# B&R Automation Studio project FlyingSaw2023
Automation Studio 4.12.2.93; technology packages: mapp 5.22.1, mappCockpit 5.22.0, mappMotion 5.22.2, mappView 5.22.1

## Configuration Config1

CPU X20CP3586, AutomationRuntime F4.93, Build 4.1.2, Safety 0.0, Vc V4.72.0

### Task classes (Cpu.sw)
```
Cyclic#1 (cycle 2000 us, tolerance 0 us):
  Saw_P <- Libraries.Saw.Saw_P.prg
  Main <- Main.prg
  ConveyorAx <- ConveyorAxis.prg
  ParallelAx <- ParallelAxis.prg
  Perpendicu <- PerpendicularAxis.prg
  Alarm <- Alarm.prg
  Recipe <- Recipe.prg
  Program <- (binary)
DataObjects: McAcpSys
NcDataObjects: McDriveLog
Binaries: udbdef, FWRules, TCData, arsvcreg, McAcpDrv, arflatprv, arcoal, McAcpSim, mvLoader, mCoWebSc, sysconf, Role, User, iomap, ashwd, asfw, arconfig, ashwac, Config_1, Config_2, Settings, Config, Config_3, McProfGen
Libraries: AsBrStr, AsTCP, standard, runtime, Saw_L, operator, McBase, CoTrace, AsZip, FileIO, MpAxis, McAxis, MpBase, McAcpAx, MpAlarmX, astime, MpServer, MpRecipe, sys_lib, asieccon, powerlnk, asepl, arssl, dataobj, aruser
```

### Hardware
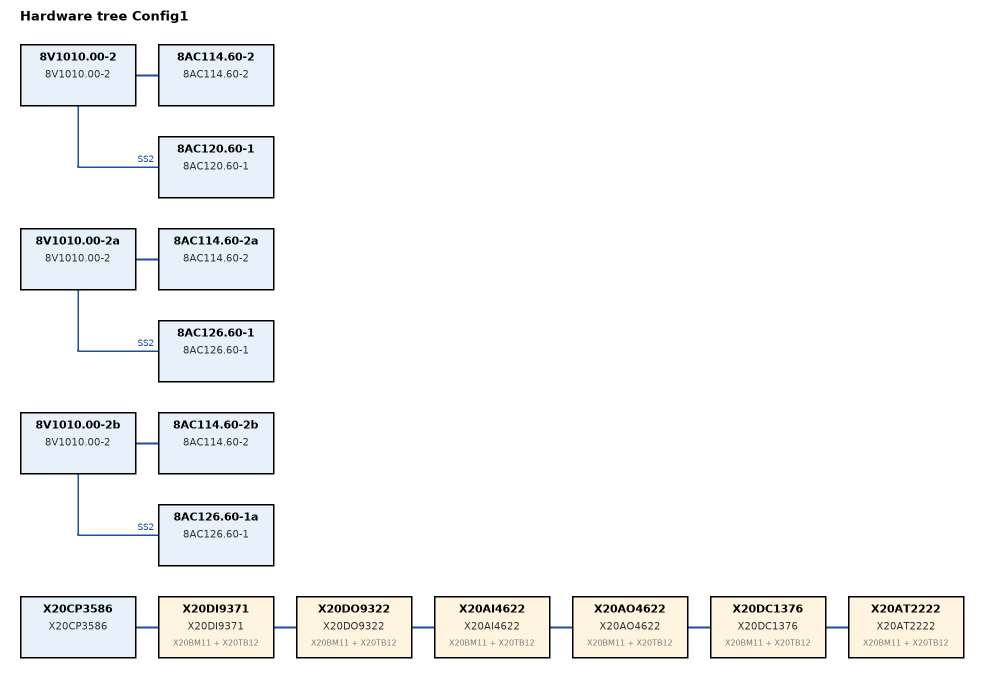
```
8AC114.60-2 : 8AC114.60-2 v1.0.0.8  [SS -> 8V1010.00-2.SS1; PLK1 -> X20CP3586.IF3 (NodeNumber=1) [Cable Type=PowerlinkCable, Length=10, Version=1.0.0.3]; PLK2 -> 8AC114.60-2a.PLK1 (NodeNumber=1) [Cable Type=PowerlinkCable, Length=10, Version=1.0.0.3]]
8AC114.60-2a : 8AC114.60-2 v1.0.0.8  [SS -> 8V1010.00-2a.SS1; PLK1 -> 8AC114.60-2.PLK2 (NodeNumber=2) [Cable Type=PowerlinkCable, Length=10, Version=1.0.0.3]; PLK2 -> 8AC114.60-2b.PLK1 (NodeNumber=2) [Cable Type=PowerlinkCable, Length=10, Version=1.0.0.3]]
8AC114.60-2b : 8AC114.60-2 v1.0.0.8  [SS -> 8V1010.00-2b.SS1; PLK1 -> 8AC114.60-2a.PLK2 (NodeNumber=3) [Cable Type=PowerlinkCable, Length=10, Version=1.0.0.3]]
8AC120.60-1 : 8AC120.60-1 v2.2.0.0  [SS -> 8V1010.00-2.SS2]
  PlugInType = Encoder
  McAcoposTypeID = AcoposPlugInConfig
8AC126.60-1 : 8AC126.60-1 v2.2.0.0  [SS -> 8V1010.00-2a.SS2]
  PlugInType = Encoder
  McAcoposTypeID = AcoposPlugInConfig
8AC126.60-1a : 8AC126.60-1 v2.2.0.0  [SS -> 8V1010.00-2b.SS2]
  PlugInType = Encoder
  McAcoposTypeID = AcoposPlugInConfig
8V1010.00-2 : 8V1010.00-2 v2.2.0.0
  DriveConfiguration/Module:
    McAcoposTypeID = AcoposConfig
    ActivateACOPOSSimulationOnPLC = 0
    PowerSupply = ETA
  DriveConfiguration/Channel[1]/RealAxis:
    AxisReference = gParallelAxis
    MechanicalElementsIsInvisible = 0
  DriveConfiguration/Channel[1]/RealAxis/MechanicalElements/Gearbox:
    InputIsReadOnly = 0
    Input = 1
    OutputIsReadOnly = 0
    Output = 1
  DriveConfiguration/Channel[1]/RealAxis/MechanicalElements/RotaryToLinearTransformation:
    ReferenceDistanceIsReadOnly = 0
    ReferenceDistance = 1.6
  DriveConfiguration/Channel[1]/RealAxis/Controller:
    ModeIsReadOnly = 0
    Mode = PositionController
  DriveConfiguration/Channel[1]/RealAxis/Controller/Mode/Position:
    ProportionalGain = 907
    IntegrationTime = 0.0
    PredictionTime = 0.0004
    TotalDelayTime = 0.0004
  DriveConfiguration/Channel[1]/RealAxis/Controller/Mode/Speed:
    ProportionalGainIsReadOnly = 0
    ProportionalGain = 0.05
    IntegrationTimeIsReadOnly = 0
    IntegrationTime = 0.0
    FilterTimeIsReadOnly = 0
    FilterTime = 0.0
  DriveConfiguration/Channel[1]/RealAxis/Controller/Mode/LoopFilters:
    LoopFilterXIsReadOnly = 0
    LoopFilter1 = NotUsed
    LoopFilter2 = NotUsed
    LoopFilter3 = NotUsed
  DriveConfiguration/Channel[1]/RealAxis/Homing:
    ModeIsReadOnly = 0
    Mode = LimitSwitch
  DriveConfiguration/Channel[1]/RealAxis/Homing/Mode:
    Position = -0.8
    StartVelocity = 0.5
    HomingVelocity = 0.05
    Acceleration = 50.0
    SwitchEdge = Negative
    HomingDirection = Positive
    KeepDirection = No
    ReferencePulse = NotUsed
  DriveConfiguration/Channel[1]/RealAxis/Homing:
    RestorePositionVariable = 
  DriveConfiguration/Channel[1]/RealAxis/StopReaction:
    QuickstopIsReadOnly = 0
    Quickstop = DecelerationLimit
    DriveErrorIsReadOnly = 0
    DriveError = DecelerationLimit
  DriveConfiguration/Channel[1]/RealAxis/MovementErrorLimits:
    PositionError = 10
    VelocityErrorMonitoring = NotUsed
  DriveConfiguration/Channel[1]/RealAxis:
    JerkFilterIsReadOnly = 0
    JerkFilter = NotUsed
    ZeroVibrationFilter = NotUsed
  DriveConfiguration/Channel[1]/RealAxis/DigitalInputs/HomingSwitch:
    SourceIsReadOnly = 0
    Source = X1Ref
    Level = High
  DriveConfiguration/Channel[1]/RealAxis/DigitalInputs/PositiveLimitSwitch:
    Source = Variable
  DriveConfiguration/Channel[1]/RealAxis/DigitalInputs/PositiveLimitSwitch/Source:
    PVmapping = ::Saw_SimInputs.diDriveParallelAtFront
  DriveConfiguration/Channel[1]/RealAxis/DigitalInputs/PositiveLimitSwitch:
    Level = High
  DriveConfiguration/Channel[1]/RealAxis/DigitalInputs/NegativeLimitSwitch:
    Source = Variable
  DriveConfiguration/Channel[1]/RealAxis/DigitalInputs/NegativeLimitSwitch/Source:
    PVmapping = ::Saw_SimInputs.diDriveParallelAtBack
  DriveConfiguration/Channel[1]/RealAxis/DigitalInputs/NegativeLimitSwitch:
    Level = High
  DriveConfiguration/Channel[1]/RealAxis/DigitalInputs/Trigger1:
    Source = X1Trigger1
    Level = High
  DriveConfiguration/Channel[1]/RealAxis/DigitalInputs/Trigger2:
    Source = X1Trigger2
    Level = High
  DriveConfiguration/Channel[1]/RealAxis/DigitalInputs/Quickstop:
    Input = Trigger2
  DriveConfiguration/Channel[1]/RealAxis/Simulation:
    SimulationModeOnPLC = SetValueGeneration
    SimulationModeOnACOPOS = NotUsed
  DriveConfiguration/Channel[1]/RealAxis/AxisFeatures:
    FeatureRef[1] = CamAutomatParallel
  DriveConfiguration/Channel[1]:
    ExternalEncoderAxis = NotUsed
8V1010.00-2a : 8V1010.00-2 v2.2.0.0
  DriveConfiguration/Module:
    McAcoposTypeID = AcoposConfig
    ActivateACOPOSSimulationOnPLC = 0
    PowerSupply = ETA
  DriveConfiguration/Channel[1]/RealAxis:
    AxisReference = gPerpendicularAxis
    MechanicalElementsIsInvisible = 0
  DriveConfiguration/Channel[1]/RealAxis/MechanicalElements/Gearbox:
    InputIsReadOnly = 0
    Input = 1
    OutputIsReadOnly = 0
    Output = 1
  DriveConfiguration/Channel[1]/RealAxis/MechanicalElements/RotaryToLinearTransformation:
    ReferenceDistanceIsReadOnly = 0
    ReferenceDistance = 1.6
  DriveConfiguration/Channel[1]/RealAxis/Controller:
    ModeIsReadOnly = 0
    Mode = PositionController
  DriveConfiguration/Channel[1]/RealAxis/Controller/Mode/Position:
    ProportionalGain = 215
    IntegrationTime = 0.0
    PredictionTime = 0.0004
    TotalDelayTime = 0.0004
  DriveConfiguration/Channel[1]/RealAxis/Controller/Mode/Speed:
    ProportionalGainIsReadOnly = 0
    ProportionalGain = 0.041
    IntegrationTimeIsReadOnly = 0
    IntegrationTime = 0.0
    FilterTimeIsReadOnly = 0
    FilterTime = 0.0
  DriveConfiguration/Channel[1]/RealAxis/Controller/Mode/LoopFilters:
    LoopFilterXIsReadOnly = 0
    LoopFilter1 = NotUsed
    LoopFilter2 = NotUsed
    LoopFilter3 = NotUsed
  DriveConfiguration/Channel[1]/RealAxis/Homing:
    ModeIsReadOnly = 0
    Mode = LimitSwitch
  DriveConfiguration/Channel[1]/RealAxis/Homing/Mode:
    Position = -0.6
    StartVelocity = 0.5
    HomingVelocity = 0.05
    Acceleration = 50.0
    SwitchEdge = Negative
    HomingDirection = Positive
    KeepDirection = No
    ReferencePulse = NotUsed
  DriveConfiguration/Channel[1]/RealAxis/Homing:
    RestorePositionVariable = 
  DriveConfiguration/Channel[1]/RealAxis/StopReaction:
    QuickstopIsReadOnly = 0
    Quickstop = DecelerationLimit
    DriveErrorIsReadOnly = 0
    DriveError = DecelerationLimit
  DriveConfiguration/Channel[1]/RealAxis/MovementErrorLimits:
    PositionError = 10
    VelocityErrorMonitoring = NotUsed
  DriveConfiguration/Channel[1]/RealAxis:
    JerkFilterIsReadOnly = 0
    JerkFilter = NotUsed
    ZeroVibrationFilter = NotUsed
  DriveConfiguration/Channel[1]/RealAxis/DigitalInputs/HomingSwitch:
    SourceIsReadOnly = 0
    Source = X1Ref
    Level = High
  DriveConfiguration/Channel[1]/RealAxis/DigitalInputs/PositiveLimitSwitch:
    Source = Variable
  DriveConfiguration/Channel[1]/RealAxis/DigitalInputs/PositiveLimitSwitch/Source:
    PVmapping = ::Saw_SimInputs.diDriveCutAtFront
  DriveConfiguration/Channel[1]/RealAxis/DigitalInputs/PositiveLimitSwitch:
    Level = High
  DriveConfiguration/Channel[1]/RealAxis/DigitalInputs/NegativeLimitSwitch:
    Source = Variable
  DriveConfiguration/Channel[1]/RealAxis/DigitalInputs/NegativeLimitSwitch/Source:
    PVmapping = ::Saw_SimInputs.diDriveCutAtBack
  DriveConfiguration/Channel[1]/RealAxis/DigitalInputs/NegativeLimitSwitch:
    Level = High
  DriveConfiguration/Channel[1]/RealAxis/DigitalInputs/Trigger1:
    Source = X1Trigger1
    Level = High
  DriveConfiguration/Channel[1]/RealAxis/DigitalInputs/Trigger2:
    Source = X1Trigger2
    Level = High
  DriveConfiguration/Channel[1]/RealAxis/DigitalInputs/Quickstop:
    Input = Trigger2
  DriveConfiguration/Channel[1]/RealAxis/Simulation:
    SimulationModeOnPLC = SetValueGeneration
    SimulationModeOnACOPOS = NotUsed
  DriveConfiguration/Channel[1]/RealAxis/AxisFeatures:
    FeatureRef[1] = CamAutomatPerpendicular
  DriveConfiguration/Channel[1]:
    ExternalEncoderAxis = NotUsed
8V1010.00-2b : 8V1010.00-2 v2.2.0.0
  DriveConfiguration/Module:
    McAcoposTypeID = AcoposConfig
    ActivateACOPOSSimulationOnPLC = 1
    PowerSupply = ETA
  DriveConfiguration/Channel[1]/RealAxis:
    AxisReference = gConveyorAxis
    MechanicalElementsIsInvisible = 0
  DriveConfiguration/Channel[1]/RealAxis/MechanicalElements/Gearbox:
    InputIsReadOnly = 0
    Input = 1
    OutputIsReadOnly = 0
    Output = 1
  DriveConfiguration/Channel[1]/RealAxis/MechanicalElements/RotaryToLinearTransformation:
    ReferenceDistanceIsReadOnly = 0
    ReferenceDistance = 1
  DriveConfiguration/Channel[1]/RealAxis/Controller:
    ModeIsReadOnly = 0
    Mode = PositionController
  DriveConfiguration/Channel[1]/RealAxis/Controller/Mode/Position:
    ProportionalGain = 50.0
    IntegrationTime = 0.0
    PredictionTime = 0.0004
    TotalDelayTime = 0.0004
  DriveConfiguration/Channel[1]/RealAxis/Controller/Mode/Speed:
    ProportionalGainIsReadOnly = 0
    ProportionalGain = 2.0
    IntegrationTimeIsReadOnly = 0
    IntegrationTime = 0.0
    FilterTimeIsReadOnly = 0
    FilterTime = 0.0
  DriveConfiguration/Channel[1]/RealAxis/Controller/Mode/LoopFilters:
    LoopFilterXIsReadOnly = 0
    LoopFilter1 = NotUsed
    LoopFilter2 = NotUsed
    LoopFilter3 = NotUsed
  DriveConfiguration/Channel[1]/RealAxis/Homing:
    ModeIsReadOnly = 0
    Mode = Direct
  DriveConfiguration/Channel[1]/RealAxis/Homing/Mode:
    Position = 0.0
    ReferencePulse = NotUsed
  DriveConfiguration/Channel[1]/RealAxis/Homing:
    RestorePositionVariable = 
  DriveConfiguration/Channel[1]/RealAxis/StopReaction:
    QuickstopIsReadOnly = 0
    Quickstop = DecelerationLimit
    DriveErrorIsReadOnly = 0
    DriveError = DecelerationLimit
  DriveConfiguration/Channel[1]/RealAxis/MovementErrorLimits:
    PositionError = 1.0
    VelocityErrorMonitoring = Automatic1
  DriveConfiguration/Channel[1]/RealAxis:
    JerkFilterIsReadOnly = 0
    JerkFilter = NotUsed
    ZeroVibrationFilter = NotUsed
  DriveConfiguration/Channel[1]/RealAxis/DigitalInputs/HomingSwitch:
    SourceIsReadOnly = 0
    Source = X1Ref
    Level = High
  DriveConfiguration/Channel[1]/RealAxis/DigitalInputs/PositiveLimitSwitch:
    Source = X1PosLim
    Level = High
  DriveConfiguration/Channel[1]/RealAxis/DigitalInputs/NegativeLimitSwitch:
    Source = X1NegLim
    Level = High
  DriveConfiguration/Channel[1]/RealAxis/DigitalInputs/Trigger1:
    Source = X1Trigger1
    Level = High
  DriveConfiguration/Channel[1]/RealAxis/DigitalInputs/Trigger2:
    Source = X1Trigger2
    Level = High
  DriveConfiguration/Channel[1]/RealAxis/DigitalInputs/Quickstop:
    Input = Trigger2
  DriveConfiguration/Channel[1]/RealAxis/Simulation:
    SimulationModeOnPLC = SetValueGeneration
    SimulationModeOnACOPOS = NotUsed
  DriveConfiguration/Channel[1]/RealAxis/AxisFeatures:
    FeatureRef[1] = Feature_CamAutomat
  DriveConfiguration/Channel[1]:
    ExternalEncoderAxis = NotUsed
X20AI4622 : X20AI4622 v1.2.0.0  [SS1 -> X20TB12b.SS; SL -> X20BM11b.SL1]
X20AO4622 : X20AO4622 v1.3.0.0  [SS1 -> X20TB12c.SS; SL -> X20BM11c.SL1]
X20AT2222 : X20AT2222 v1.4.0.0  [SS1 -> X20TB12e.SS; SL -> X20BM11e.SL1]
X20BM11 : X20BM11 v1.1.0.0  [X2X1 -> X20CP3586.IF6]
X20BM11a : X20BM11 v1.1.0.0  [X2X1 -> X20BM11.X2X2]
X20BM11b : X20BM11 v1.1.0.0  [X2X1 -> X20BM11a.X2X2]
X20BM11c : X20BM11 v1.1.0.0  [X2X1 -> X20BM11b.X2X2]
X20BM11d : X20BM11 v1.1.0.0  [X2X1 -> X20BM11c.X2X2]
X20BM11e : X20BM11 v1.1.0.0  [X2X1 -> X20BM11d.X2X2]
X20CP3586 : X20CP3586 v1.10.0.0
  Connector IF2:
    ActivateDevice = 1
    Mode = Manual
    InternetAddress = 10.0.0.2
    SubnetMask = 255.255.255.0
    ActivateSnmp = 2
  Connector IF3:
    DNAConfiguration = manual
    Channel1
    ChannelID1 = McAcpBroadcast
    ChannelType1 = OCTET[96]
  ConfigurationID = FlyingSaw2023_Config1
  UserPartitionSize = 0
  Simulation = 1
  TimerDeviceType = EPLX2X
  TimerDevice = X20CP3586.IF3
  TaskClassIdleTime = 2000
  Cyclic1Duration = 2000
  Cyclic1Tolerance = 0
  FileDevice1
  FileDeviceName1 = USER
  FileDevicePath1 = C:\temp
  ActivateOpcUa = 1
  OpcUaInformationModels_PV_Version = 1
X20DC1376 : X20DC1376 v1.3.0.0  [SS1 -> X20TB12d.SS; SL -> X20BM11d.SL1]
X20DI9371 : X20DI9371 v1.4.0.0  [SS1 -> X20TB12.SS; SL -> X20BM11.SL1]
X20DO9322 : X20DO9322 v1.5.0.0  [SS1 -> X20TB12a.SS; SL -> X20BM11a.SL1]
X20TB12 : X20TB12 v1.0.0.0
X20TB12a : X20TB12 v1.0.0.0
X20TB12b : X20TB12 v1.0.0.0
X20TB12c : X20TB12 v1.0.0.0
X20TB12d : X20TB12 v1.0.0.0
X20TB12e : X20TB12 v1.0.0.0
```

### IoMap.iom - X20CP3586/IoMap.iom
```iecst
VAR_CONFIG
	::Main:SawLeft AT %IX."X20DI9371".DigitalInput01;
	::Main:SawRight AT %IX."X20DI9371".DigitalInput02;
	::Main:SawRunAxis AT %IX."X20DI9371".DigitalInput06;
	::Tasmociag:MpAxisConveyor.MoveVelocity AT %QX."X20DO9322".DigitalOutput01;
	::Main:RunConveyor AT %IX."X20DI9371".DigitalInput05;
	::Main:SawForward AT %IX."X20DI9371".DigitalInput03;
	::Main:SawBackward AT %IX."X20DI9371".DigitalInput04;
	::OsRownoleg:MpAxisParallel.Power AT %QX."X20DO9322".DigitalOutput02;
	::OsRownoleg:MpAxisParallel.Power AT %QX."X20DO9322".DigitalOutput03;
END_VAR
```

### Config_1.axis - X20CP3586/mappMotion/Config_1.axis
```
Element gPerpendicularAxis (Type=axis)
  BaseTypeIsReadOnly = 0
  BaseType = LinearBounded
    MeasurementUnit = 5067858
    MeasurementResolutionIsReadOnly = 0
    MeasurementResolution = 0.001
    CountDirectionIsReadOnly = 0
    CountDirection = Standard
  MovementLimitsIsReadOnly = 0
  MovementLimits = Internal
    Position:
      LowerLimitMin = -1.79769313486231E308
      UpperLimitMax = 1.79769313486231E308
      LowerLimit = -0.6
      UpperLimit = 1.2
    VelocityIsReadOnly = 0
    Velocity:
      VelocityMax = 3.4E38
      Velocity = 50
    AccelerationIsReadOnly = 0
    Acceleration:
      AccelerationMax = 3.4E38
      Acceleration = 3000
    DecelerationIsReadOnly = 0
    Deceleration:
      DecelerationMax = 3.4E38
      Deceleration = 3000
  Alarms = MpAlarmX
    mapp.AlarmX.Core.Configuration:
      [0]:
        Message = System problem on Perpendicular axis
        Code = 1001
        Severity = 50
      [1]:
        Message = Initialization problem on Perpendicular axis
        Code = 1002
        Severity = 10
      [2]:
        Message = Parameter problem on Perpendicular axis
        Code = 1003
        Severity = 10
      [3]:
        Message = Operation problem on Perpendicular axis
        Code = 1004
        Severity = 30
      [4]:
        Message = Data access problem on Perpendicular axis
        Code = 1005
        Severity = 10
      [5]:
        Message = Syntax error on Perpendicular axis
        Code = 1006
        Severity = 10
      [9]:
        Message = Network problem on Perpendicular axis
        Code = 1007
        Severity = 10
      [10]:
        Message = Encoder problem on Perpendicular axis
        Code = 1008
        Severity = 30
      [11]:
        Message = Drive problem on Perpendicular axis
        Code = 1009
        Severity = 30
      [12]:
        Message = IO problem on Perpendicular axis
        Code = 1010
        Severity = 20
      [13]:
        Message = Supply problem on Perpendicular axis
        Code = 1011
        Severity = 10
      [14]:
        Message = Motor problem on Perpendicular axis
        Code = 1012
        Severity = 50
      [15]:
        Message = Holding brake problem on Perpendicular axis
        Code = 1013
        Severity = 50
      [19]:
        Message = Movement error limit reached on Perpendicular axis on Perpendicular axis
        Code = 1014
        Severity = 40
      [20]:
        Message = HW or SW movement limits reached on Perpendicular axis on Perpendicular axis
        Code = 1015
        Severity = 40
      [21]:
        Message = Enable input low on Perpendicular axis
        Code = 1016
        Severity = 10
Element gParallelAxis (Type=axis)
  BaseTypeIsReadOnly = 0
  BaseType = LinearBounded
    MeasurementUnit = 5067858
    MeasurementResolutionIsReadOnly = 0
    MeasurementResolution = 0.001
    CountDirectionIsReadOnly = 0
    CountDirection = Standard
  MovementLimitsIsReadOnly = 0
  MovementLimits = Internal
    Position:
      LowerLimitMin = -1.79769313486231E308
      UpperLimitMax = 1.79769313486231E308
      LowerLimit = -0.8
      UpperLimit = 0.8
    VelocityIsReadOnly = 0
    Velocity:
      VelocityMax = 3.4E38
      Velocity = 50
    AccelerationIsReadOnly = 0
    Acceleration:
      AccelerationMax = 3.4E38
      Acceleration = 3000
    DecelerationIsReadOnly = 0
    Deceleration:
      DecelerationMax = 3.4E38
      Deceleration = 3000
  Alarms = MpAlarmX
    mapp.AlarmX.Core.Configuration:
      [0]:
        Code = 2001
        Severity = 50
      [1]:
        Message = Initialization problem on parallel axis
        Code = 2002
        Severity = 10
      [2]:
        Message = Parameter problem on parallel axis
        Code = 2003
        Severity = 10
      [3]:
        Message = Operation problem on parallel axis
        Code = 2004
        Severity = 30
      [4]:
        Message = Data access problem on parallel axis
        Code = 2005
        Severity = 10
      [5]:
        Message = Syntax error on parallel axis
        Code = 2006
        Severity = 10
      [9]:
        Message = Network problem on parallel axis
        Code = 2007
        Severity = 10
      [10]:
        Message = Encoder problem on parallel axis
        Code = 2008
        Severity = 30
      [11]:
        Message =  on parallel axis
        Code = 2009
        Severity = 20
      [12]:
        Message = IO problem on parallel axis
        Code = 2010
        Severity = 10
      [13]:
        Message = Supply problem on parallel axis
        Code = 2011
        Severity = 10
      [14]:
        Message = Motor problem on parallel axis
        Code = 2012
        Severity = 50
      [15]:
        Message = Holding brake problem on parallel axis
        Code = 2013
        Severity = 50
      [19]:
        Message = Movement error limit reached on parallel axis
        Code = 2014
        Severity = 30
      [20]:
        Message = HW or SW movement limits reached on parallel axis
        Code = 2015
        Severity = 30
      [21]:
        Message = Enable input low on parallel axis
        Code = 2016
        Severity = 10
Element gConveyorAxis (Type=axis)
  BaseTypeIsReadOnly = 0
  BaseType = LinearBounded
    MeasurementUnit = 5067858
    MeasurementResolutionIsReadOnly = 0
    MeasurementResolution = 0.001
    CountDirectionIsReadOnly = 0
    CountDirection = Standard
  MovementLimitsIsReadOnly = 0
  MovementLimits = Internal
    Position:
      LowerLimitMin = -1.79769313486231E308
      UpperLimitMax = 1.79769313486231E308
      LowerLimit = -1000.0
      UpperLimit = 5000
    VelocityIsReadOnly = 0
    Velocity:
      VelocityMax = 3.4E38
      Velocity = 10.0
    AccelerationIsReadOnly = 0
    Acceleration:
      AccelerationMax = 3.4E38
      Acceleration = 50.0
    DecelerationIsReadOnly = 0
    Deceleration:
      DecelerationMax = 3.4E38
      Deceleration = 50.0
  Alarms = MpAlarmX
    mapp.AlarmX.Core.Configuration:
      [0]:
        Message = System problem on Convoyer axis
        Code = 3001
        Severity = 50
      [1]:
        Message = Initialization problem on Convoyer axis
        Code = 3002
        Severity = 10
      [2]:
        Message = Parameter problem on Convoyer axis
        Code = 3003
        Severity = 10
      [3]:
        Message = Operation problem on Convoyer axis
        Code = 3004
        Severity = 30
      [4]:
        Message = Data access problem on Convoyer axis
        Code = 3005
        Severity = 10
      [5]:
        Message = Syntax error on Convoyer axis
        Code = 3006
        Severity = 10
      [9]:
        Message = Network problem on Convoyer axis
        Code = 3007
        Severity = 10
      [10]:
        Message = Encoder problem on Convoyer axis
        Code = 3008
        Severity = 30
      [11]:
        Message = Drive problem on Convoyer axis
        Code = 3009
        Severity = 30
      [12]:
        Message = IO problem on Convoyer axis
        Code = 3010
        Severity = 20
      [13]:
        Message = Supply problem on Convoyer axis
        Code = 3011
        Severity = 10
      [14]:
        Message = Motor problem on Convoyer axis
        Code = 3012
        Severity = 50
      [15]:
        Message = Holding brake problem on Convoyer axis
        Code = 3013
        Severity = 50
      [19]:
        Message = Movement error limit reached on Convoyer axis
        Code = 3014
        Severity = 30
      [20]:
        Message = HW or SW movement limits reached on Convoyer axis
        Code = 3015
        Severity = 30
      [21]:
        Message = Enable input low on Convoyer axis
        Code = 3016
        Severity = 10
```

### Config_2.axisfeature - X20CP3586/mappMotion/Config_2.axisfeature
```
Element CamAutomatParallel (Type=axisfeature)
  Type = CamAutomat
    CamAutomatType = ACOPOS
      CommonParameters:
        Master:
          ValueSource = SetPosition
            AxisReference = gConveyorAxis
            MaxVelocity = 1.0
          StartPosition = 0.0
          StartInterval = MasterAxisPeriod
        AdvancedParameters:
          StartStateParameters:
            StartState = 0
            RelMasterStartPos = 0.0
          AdditiveAxes:
            AdditiveMasterValueSource = NotUsed
            AdditiveSlaveValueSource = NotUsed
          MasterStartPositionMode = NotEvaluatedAnew
          ControlSettings:
            CrossLeftBoundary = PositionLimitedHorizontal
            CamChangeImmediately = CurrentMasterMoveDir
          MessageSettings:
            ErrorsInStandby = NoErrorMessages
          TriggerAndLatch:
            Trigger1Delay = 0.0
            Trigger2Delay = 0.0
            SlaveLatchParID = 0
          EventParIDs
          StartIntervals
          Factors:
            SlaveFactorParID = 0
      States:
        State0 = Used
          Events:
            Event[0]:
              Type = StateEnd
              Transition = EndOfState
              SynchronousUpdate = NotUsed
              NextState = 1
        State[1]:
          Cam = Predefined
            PredefinedCam = OneToOne
          MasterFactor = 300
          SlaveFactor = 300
          CompensationMode = DistancesBetweenExitEntryPoints
            MasterDistance = 0.2
            SlaveDistance = 0.2
            AdvancedParameters = NotUsed
          AdvancedParameters:
            RepeatCounterInit = 0
            MasterValueSource = CommonMaster
          Events:
            Event[0]:
              Type = StateEnd
              Transition = EndOfState
              SynchronousUpdate = NotUsed
              NextState = 2
        State[2]:
          Cam = Predefined
            PredefinedCam = OneToOne
          MasterFactor = 300
          SlaveFactor = -300
          CompensationMode = DistancesBetweenExitEntryPoints
            MasterDistance = 0.2
            SlaveDistance = -0.2
            AdvancedParameters = NotUsed
          AdvancedParameters:
            RepeatCounterInit = 0
            MasterValueSource = CommonMaster
          Events:
            Event[0]:
              Type = Signal1FromPLC
              Transition = EndOfState
              SynchronousUpdate = NotUsed
              NextState = 255
            Event[1]:
              Type = StateEnd
              Transition = EndOfState
              SynchronousUpdate = NotUsed
              NextState = 1
Element CamAutomatPerpendicular (Type=axisfeature)
  Type = CamAutomat
    CamAutomatType = ACOPOS
      CommonParameters:
        Master:
          ValueSource = SetPosition
            AxisReference = gConveyorAxis
            MaxVelocity = 1.0
          StartPosition = 0.0
          StartInterval = MasterAxisPeriod
        AdvancedParameters:
          StartStateParameters:
            StartState = 0
            RelMasterStartPos = 0.0
          AdditiveAxes:
            AdditiveMasterValueSource = NotUsed
            AdditiveSlaveValueSource = NotUsed
          MasterStartPositionMode = NotEvaluatedAnew
          ControlSettings:
            CrossLeftBoundary = PositionLimitedHorizontal
            CamChangeImmediately = CurrentMasterMoveDir
          MessageSettings:
            ErrorsInStandby = NoErrorMessages
          TriggerAndLatch:
            Trigger1Delay = 0.0
            Trigger2Delay = 0.0
            SlaveLatchParID = 0
          EventParIDs
          StartIntervals
          Factors:
            SlaveFactorParID = 0
      States:
        State0 = Used
          Events:
            Event[0]:
              Type = StateEnd
              Transition = EndOfState
              SynchronousUpdate = NotUsed
              NextState = 1
        State[1]:
          Cam = Predefined
            PredefinedCam = OneToOne
          MasterFactor = 125
          SlaveFactor = 200
          CompensationMode = DistancesBetweenExitEntryPoints
            MasterDistance = 0.125
            SlaveDistance = 0.3
            AdvancedParameters = NotUsed
          AdvancedParameters:
            RepeatCounterInit = 0
            MasterValueSource = CommonMaster
          Events:
            Event[0]:
              Type = StateEnd
              Transition = EndOfState
              SynchronousUpdate = NotUsed
              NextState = 2
        State[2]:
          Cam = Predefined
            PredefinedCam = OneToOne
          MasterFactor = 125
          SlaveFactor = -200
          CompensationMode = DistancesBetweenExitEntryPoints
            MasterDistance = 0.125
            SlaveDistance = -0.3
            AdvancedParameters = NotUsed
          AdvancedParameters:
            RepeatCounterInit = 0
            MasterValueSource = CommonMaster
          Events:
            Event[0]:
              Type = StateEnd
              Transition = EndOfState
              SynchronousUpdate = NotUsed
              NextState = 3
        State[3]:
          Cam = Predefined
            PredefinedCam = OneToOne
          MasterFactor = 500
          SlaveFactor = 0
          CompensationMode = NoCompensation
          AdvancedParameters:
            RepeatCounterInit = 0
            MasterValueSource = CommonMaster
          Events:
            Event[0]:
              Type = Signal1FromPLC
              Transition = EndOfState
              SynchronousUpdate = NotUsed
              NextState = 255
            Event[1]:
              Type = StateEnd
              Transition = EndOfState
              SynchronousUpdate = NotUsed
              NextState = 1
```

### Config.mpalarmxcore - X20CP3586/mappServices/Config.mpalarmxcore
```
Element gAlarmXCore (Type=mpalarmxcore)
  mapp.AlarmX.Core.Configuration:
    [0]:
      Name = SpeedToHigh
      Message = Convoyer speed set to high
      Code = 3101
      Severity = 30
      Behavior = LevelMonitoring
        Monitoring:
          MonitoredPV = ::Main:ConveyorSpeed
          HighLimitEnable = Static
            Limit = 100
    [1]:
      Name = Wrong parallel step
      Message = Wrong parallel step
      Code = 2101
      Severity = 20
      Behavior = LevelMonitoring
        Monitoring:
          MonitoredPV = ::Main:ParallelStep
          LowLimitEnable = Static
            Limit = 0
          HighLimitEnable = Static
            Limit = 1.6
    [2]:
      Name = Wrong perpendicular step
      Message = Wrong perpendicular step
      Code = 1101
      Severity = 20
      Behavior = LevelMonitoring
        Monitoring:
          MonitoredPV = ::Main:PerpendicularStep
          LowLimitEnable = Static
          HighLimitEnable = Static
            Limit = 2
    [3]:
      Name = Dangerous feed rate
      Message = This setting may harm the machine
      Code = 1102
      Severity = 50
      Behavior = LevelMonitoring
        Monitoring:
          MonitoredPV = ::gPerpendicularSettings.FeedRate
          LowLimitEnable = Static
            Limit = 2
          HighLimitEnable = Static
            Limit = 3
    [4]:
      Name = Dangerous torque
      Message = This setting may harm the machine
      Code = 1103
      Severity = 50
      Behavior = LevelMonitoring
        Monitoring:
          HighLimitEnable = Static
            Limit = 20
    [5]:
      Name = Dangerous log length
      Message = This setting may harm the machine
      Code = 1104
      Severity = 50
      Behavior = LevelMonitoring
        Monitoring:
          LowLimitEnable = Static
            Limit = 1
```

### Config_4.mprecipexml - X20CP3586/mappServices/Config_4.mprecipexml
```
Element gRecipeXml (Type=mprecipexml)
  Alarms = MpAlarmX
Element gRecipeXml_1 (Type=mprecipexml)
Element gRecipeXml_2 (Type=mprecipexml)
  Alarms = MpAlarmX
    mapp.AlarmX.Core.Configuration:
      [0]:
        Code = 4001
        Severity = 20
      [1]:
        Code = 4002
        Severity = 10
      [2]:
        Code = 4003
        Severity = 50
      [3]:
        Code = 4004
        Severity = 40
```

## Logical view

Binary libraries used (declarations not repeated): operator, standard, runtime, astime, AsBrStr, AsTCP, AsIecCon, McBase, CoTrace, AsZip, FileIO, MpAxis, McAxis, MpBase, McAcpAx, MpAlarmX, MpServer, MpRecipe, sys_lib

### Global.typ - Global data types
```iecst
TYPE
	gRecipeMenagmentType : 	STRUCT
		Load1M : BOOL;
		Save1M : BOOL;
		Save2M : BOOL;
		Load2M : BOOL;
		Save3M : BOOL;
		Load3M : BOOL;
	END_STRUCT;
	gConvoyerSettingsType : 	STRUCT
		doReadyToWork : BOOL;
		diRun : BOOL;
		aiSpeed : REAL;
	END_STRUCT;
	gOperatingPanelTyp : 	STRUCT
		diStart : BOOL;
		diHomeParallel : BOOL;
		diHomePerpendicular : BOOL;
		StartSequence : BOOL;
		StopSequence : BOOL;
		SwitchModeToAuto : BOOL;
		SwitchModeToMan : BOOL;
		LoadRecipe1M : BOOL;
		LoadRecipe2M : BOOL;
		LoadRecipe3M : BOOL;
		SaveRecipe1M : BOOL;
		SaveRecipe2M : BOOL;
		SaveRecipe3M : BOOL;
	END_STRUCT;
	gParallelSettingsType : 	STRUCT
		doReadyToWork : BOOL;
		aiParallelStep : REAL;
		diRight : BOOL;
		diLeft : BOOL;
		AutoReady : BOOL;
		ReadyToChange : BOOL;
		AfterSwitchFlag : BOOL;
	END_STRUCT;
	gPerpendicularSettingsType : 	STRUCT
		doReadyToWork : BOOL;
		aiPerpendicularStep : REAL;
		diForward : BOOL;
		diBackward : BOOL;
		AutoReady : BOOL;
		ReadyToChange : BOOL;
		AfterSwitchFlag : BOOL;
		AccTorque : REAL;
		WoodLogLength : REAL;
		FeedRate : REAL;
	END_STRUCT;
	gRecipe1MTyp : 	STRUCT
		WoodLogLength : REAL := 1;
		AccTorqueLimit : REAL := 10;
		SawFeedRate : REAL := 3;
	END_STRUCT;
	gRecipe2MTyp : 	STRUCT
		WoodLogLength : REAL := 2;
		AccTorqueLimit : REAL := 10;
		SawFeedRate : REAL := 3;
	END_STRUCT;
	gRecipe3MTyp : 	STRUCT
		WoodLogLength : REAL := 3;
		AccTorqueLimit : REAL := 10;
		SawFeedRate : REAL := 3;
	END_STRUCT;
END_TYPE
```

### Global.var - Global variables
```iecst
VAR
	gRecipeMenagement : gRecipeMenagmentType;
	gResetErrors : BOOL;
	gInitProgressBarValue : USINT;
	gOperatingPanel : gOperatingPanelTyp;
	gStateSetter : INT;
	gConveyorSettings : gConvoyerSettingsType;
	gPerpendicularSettings : gPerpendicularSettingsType;
	gSawOn : BOOL;
	gParallelSettings : gParallelSettingsType;
	gRecipe1M : gRecipe1MTyp;
	gRecipe2M : gRecipe2MTyp;
	gRecipe3M : gRecipe3MTyp;
END_VAR
```

### Package Logical/Libraries - Global libraries

### Library Logical/Libraries/Saw/Saw_L (ANSIC)
Depends on: AsTCP, operator, runtime, astime, standard, AsArLog, AsBrStr, Convert

#### MNG_ComHdlr.hpp
```cpp
#ifndef _MNGCOMHDLR_HPP_
#define _MNGCOMHDLR_HPP_

#define TRUE  1
#define FALSE 0

#include "MNG_InternalTyp.hpp"

#include <bur/plc.h>
#include <bur/plctypes.h>
#include <AsTCP.h>
#include <standard.h>
#include <astime.h>
#include <runtime.h>
#include <AsBrStr.h>

typedef struct{
	TcpOpen_typ tcpOpen;
	TcpIoctl_typ tcpIoctl;
	tcpLINGER_typ tcpLINGER;
	TcpSend_typ tcpSend;
	TcpClose_typ tcpClose;
	TcpRecv_typ tcpRecv;
	TcpClient_typ tcpClient;
} asTcpFcn_t;

typedef enum {
	MNG_wSock,
	MNG_skippedMessage
} MNG_errorCases;

typedef enum {
	MNG_Init,
	MNG_Socket,
	MNG_Open,
	MNG_SetIo,
	MNG_Linger,
	MNG_Connecting,
	MNG_Exchange,
	MNG_Closing,
        MNG_Reset
} MNG_internalState_t;

	extern unsigned long int MNG_CpyOutToMsg(MNG_RawDatagram * pToServer, unsigned long int counter, Saw_OUTPUTS_32BIT_FWRD *pSimOutputs);
	extern unsigned long int MNG_CpyMsgToInp(MNG_RawDatagram * pFromServer, Saw_INPUTS_32BIT_FWRD *pSimInputs);

class MNG_ComHdlr
{
	public:

	MNG_ComHdlr(char *srvIpAdr, unsigned int srvPort, TIME sendCycleTime);
	~MNG_ComHdlr();

	int RunCommunication(void*, void*, BOOL*);

	private:

	char* _srvIpAdr;
	unsigned int _srvPort;
	TIME _sendCycleTime;

	unsigned int _error;

	MNG_internalState_t _internalState;
	TON_typ _connectionTon;
	TIME _connectionTime;

	bool _connect;
	bool _sendDone;

	signed int _recvOffset;

	signed long int _potMsgLen;
	signed long int _totalRecvLen;

	unsigned long int _one;
	unsigned long int _counter;
	unsigned long int _recvLen;
	unsigned long int _recvBuffer[10000];
	TON_typ _sendTon;
	unsigned int cnt;
	MNG_RawDatagram _recvMessage;
	MNG_RawDatagram _sendMessage;

	static const signed long int SIXTEEN = 16;
	static const unsigned int PORT = 0;
	static const unsigned long int MNG_MAXPAYLOAD = 1400;

	void init_TcpOpen();
	void init_TcpSocket();
	void init_TcpIoctl();
	void init_TcpLinger();
	void init_TcpClient();
	void init_TcpRecv();
	void init_TcpSend(Saw_OUTPUTS_32BIT_FWRD* pSimOut);

	void InitParams();

	void SetSendDone(bool toogle);
	void SetStateValue(MNG_internalState_t stateVal);

};
#endif
```

#### MNG_ComHdlr.cpp
```cpp
#include "MNG_ComHdlr.hpp"
#include "MNG_CpyMsgToInp.cpp"
#include "MNG_CpyOutToMsg.cpp"

asTcpFcn_t _asTcpFcn;

MNG_ComHdlr::MNG_ComHdlr(char *srvIpAdr, unsigned int srvPort, TIME sendCycleTime)
{
	_srvIpAdr = srvIpAdr;
	_srvPort = srvPort;
	_sendCycleTime = sendCycleTime;
	InitParams();
}

MNG_ComHdlr::~MNG_ComHdlr()
{
}

int MNG_ComHdlr::RunCommunication(void* pSimInputs, void* pSimOutputs, BOOL* pSimActive) {

        unsigned long int _lastCounter = _counter;

	Saw_INPUTS_32BIT_FWRD* pFwrd_SimInputs = static_cast<Saw_INPUTS_32BIT_FWRD*>((pSimInputs));
	Saw_OUTPUTS_32BIT_FWRD* pFwrd_SimOutputs = static_cast<Saw_OUTPUTS_32BIT_FWRD*>((pSimOutputs));

	switch (_internalState) {

		case MNG_Init:
                        *pSimActive = FALSE;
			_asTcpFcn.tcpOpen.enable = FALSE;
			TcpOpen(&_asTcpFcn.tcpOpen);
			_asTcpFcn.tcpIoctl.enable = FALSE;
			TcpIoctl(&_asTcpFcn.tcpIoctl);
			_asTcpFcn.tcpClient.enable = FALSE;
			TcpClient(&_asTcpFcn.tcpClient);
			_asTcpFcn.tcpSend.enable = FALSE;
			TcpSend(&_asTcpFcn.tcpSend);
			_asTcpFcn.tcpRecv.enable = FALSE;
			TcpRecv(&_asTcpFcn.tcpRecv);
			_asTcpFcn.tcpClose.enable = FALSE;
			TcpClose(&_asTcpFcn.tcpClose);

			_connectionTon.IN = FALSE;
			_connectionTon.PT = _connectionTime;
			_sendTon.IN = FALSE;
			_sendTon.PT = _sendCycleTime;
			SetStateValue(MNG_Socket);
			break;

		case MNG_Socket:
                        *pSimActive = FALSE;
			init_TcpSocket();
			TcpOpen(&_asTcpFcn.tcpOpen);
			_recvOffset = 0;
			if (_connect == 1) {
				SetStateValue(MNG_Open);
				_connectionTon.IN = FALSE;
			}
			break;

		case MNG_Open:
                        *pSimActive = FALSE;
			init_TcpOpen();
			TcpOpen(&_asTcpFcn.tcpOpen);
			if (_asTcpFcn.tcpOpen.status == 0) {
				SetStateValue(MNG_Linger);
				_asTcpFcn.tcpIoctl.enable = FALSE;
				TcpIoctl(&_asTcpFcn.tcpIoctl);
				_connectionTon.IN = FALSE;
			}
			break;

		case MNG_SetIo:
                        *pSimActive = FALSE;
			init_TcpIoctl();
			TcpIoctl(&_asTcpFcn.tcpIoctl);
			if (_asTcpFcn.tcpIoctl.status == 0) {
				SetStateValue(MNG_Linger);
				_asTcpFcn.tcpClient.enable = FALSE;
				TcpClient(&_asTcpFcn.tcpClient);
				_connectionTon.IN = FALSE;
			}
			break;

		case MNG_Linger:
                        *pSimActive = FALSE;
			init_TcpLinger();
			TcpIoctl(&_asTcpFcn.tcpIoctl);

			if (_asTcpFcn.tcpIoctl.status == 0) {
				SetStateValue(MNG_Connecting);
				_asTcpFcn.tcpClient.enable = FALSE;
				_connectionTon.IN = FALSE;
			}

		case MNG_Connecting:
                        *pSimActive = FALSE;
			_asTcpFcn.tcpClient.enable = TRUE;
			_asTcpFcn.tcpClient.ident = _asTcpFcn.tcpOpen.ident;
			_asTcpFcn.tcpClient.portserv = _srvPort;
			_asTcpFcn.tcpClient.pServer = (long)_srvIpAdr;
			TcpClient(&_asTcpFcn.tcpClient);

			if (_asTcpFcn.tcpClient.status == ERR_FUB_BUSY) {
				// state = state || SetStateValue(Connecting);
			} else if (_asTcpFcn.tcpClient.status == 0) {
				SetStateValue(MNG_Exchange);
				_connectionTon.IN = FALSE;
				SetSendDone(TRUE);
			}
			break;

		case MNG_Exchange:
			init_TcpRecv();
			TcpRecv(&_asTcpFcn.tcpRecv);

			if (_asTcpFcn.tcpRecv.status==0){
                        *pSimActive = FALSE;
			_connectionTon.IN = FALSE;
			_recvLen = _asTcpFcn.tcpRecv.recvlen;
			_potMsgLen = N_TO_HUDINT(_recvBuffer[3]) + SIXTEEN;
			_totalRecvLen = _recvOffset + _recvLen;

			if ((_totalRecvLen < SIXTEEN) || (_totalRecvLen < _potMsgLen)) {
			_recvOffset = _recvOffset + _recvLen;
			}	else {
			while ((_potMsgLen > 0) && (_potMsgLen <= _totalRecvLen)) {
			// misconfigured message sizes
                        if ((unsigned long int)_potMsgLen > sizeof(_recvMessage)) {
			SetStateValue(MNG_Reset);
			break;
			}

			brsmemcpy((unsigned long int) &_recvMessage, (unsigned long int) &_recvBuffer, _potMsgLen*sizeof(unsigned long int));
			_totalRecvLen = _totalRecvLen - _potMsgLen;
			brsmemmove((unsigned long int) &_recvBuffer, (unsigned long int) &_recvBuffer + _potMsgLen, _totalRecvLen*sizeof(unsigned long int));
			_counter = MNG_CpyMsgToInp(&_recvMessage,pFwrd_SimInputs);
                        *pSimActive = (_lastCounter != _counter);
			_recvOffset = _totalRecvLen;

			if (_totalRecvLen > SIXTEEN) {
			_potMsgLen = N_TO_HUDINT(_recvBuffer[3]) + SIXTEEN;
			} else {
			_potMsgLen = 0;
			}

			}
			}
			}

			_sendTon.IN = _sendDone;
			TON(&_sendTon);

			if (_sendTon.Q || _asTcpFcn.tcpSend.enable == 1) {
				if (_sendDone==TRUE) {
					SetSendDone(FALSE);
					MNG_CpyOutToMsg(&_sendMessage, _counter,pFwrd_SimOutputs);
					init_TcpSend(pFwrd_SimOutputs);
				}
				TcpSend(&_asTcpFcn.tcpSend);

				if (_asTcpFcn.tcpSend.status == 0) {
					if (_asTcpFcn.tcpSend.datalen != _asTcpFcn.tcpSend.sentlen) {
						// state = state || SetStateValue(Exchange);
					}
					_asTcpFcn.tcpSend.enable = FALSE;
					SetSendDone(TRUE);
				}
			}
			if (_asTcpFcn.tcpRecv.status == tcpERR_NOT_CONNECTED) {
				SetStateValue(MNG_Closing);
			}
			break;

		case MNG_Closing:
                        *pSimActive = FALSE;
			_asTcpFcn.tcpClose.enable = TRUE;
			_asTcpFcn.tcpClose.ident = _asTcpFcn.tcpOpen.ident;
			_asTcpFcn.tcpClose.how = 0;
			TcpClose(&_asTcpFcn.tcpClose);

			if(_asTcpFcn.tcpClose.status == 0 || _asTcpFcn.tcpClose.status == 32600){
				SetStateValue(MNG_Init);
			}
			break;

                case MNG_Reset:
                        SetStateValue(MNG_Closing);
                        break;
	}

	TON(&_connectionTon);
	_connectionTon.IN = TRUE;
	if (_connectionTon.Q == 1) {
		SetStateValue(MNG_Closing);
		_connectionTon.IN = FALSE;
	}

	return _internalState;
}

void MNG_ComHdlr::init_TcpOpen(){
	_asTcpFcn.tcpOpen.enable = _connect;
}

void MNG_ComHdlr::init_TcpSocket(){
	_asTcpFcn.tcpOpen.enable = TRUE;
	_asTcpFcn.tcpOpen.pIfAddr = 0;
	_asTcpFcn.tcpOpen.port = PORT;
	_asTcpFcn.tcpOpen.options = tcpOPT_REUSEADDR;
}

void MNG_ComHdlr::init_TcpIoctl(){
	_asTcpFcn.tcpIoctl.enable = TRUE;
	_asTcpFcn.tcpIoctl.pData = (unsigned long int) &_one;
	_asTcpFcn.tcpIoctl.datalen = 4;
	_asTcpFcn.tcpIoctl.ident = _asTcpFcn.tcpOpen.ident;
	_asTcpFcn.tcpIoctl.ioctl = tcpTCP_NODELAY_SET;
}

void MNG_ComHdlr::init_TcpLinger(){
	_asTcpFcn.tcpLINGER.lLinger = FALSE;
	_asTcpFcn.tcpLINGER.lOnOff = TRUE;
	_asTcpFcn.tcpIoctl.enable = TRUE;
	_asTcpFcn.tcpIoctl.pData = (unsigned long int) &_asTcpFcn.tcpLINGER;
	_asTcpFcn.tcpIoctl.datalen = sizeof(_asTcpFcn.tcpLINGER);
	_asTcpFcn.tcpIoctl.ident = _asTcpFcn.tcpOpen.ident;
	_asTcpFcn.tcpIoctl.ioctl = tcpSO_LINGER_SET;
}

void MNG_ComHdlr::init_TcpClient(){

	_asTcpFcn.tcpClient.enable = TRUE;
	_asTcpFcn.tcpClient.ident = _asTcpFcn.tcpOpen.ident;
	_asTcpFcn.tcpClient.portserv = _srvPort;
	_asTcpFcn.tcpClient.pServer = (long)_srvIpAdr;
}

void MNG_ComHdlr::init_TcpRecv(){

	_asTcpFcn.tcpRecv.enable = TRUE;
	_asTcpFcn.tcpRecv.ident= _asTcpFcn.tcpOpen.ident;
	_asTcpFcn.tcpRecv.datamax = sizeof(_recvBuffer) - _recvOffset;
	_asTcpFcn.tcpRecv.pData = (unsigned long int) &_recvBuffer + _recvOffset;
}

void MNG_ComHdlr::init_TcpSend(Saw_OUTPUTS_32BIT_FWRD *pSimOutputs){

	_asTcpFcn.tcpSend.enable = TRUE;
	_asTcpFcn.tcpSend.ident= _asTcpFcn.tcpOpen.ident;
	_asTcpFcn.tcpSend.datalen = 16 + ((pSimOutputs->NumSignals) + 1) * 4;
	_asTcpFcn.tcpSend.pData = (unsigned long int)&_sendMessage;
	_asTcpFcn.tcpSend.flags = 0;
}

void MNG_ComHdlr::InitParams(){
	_internalState = MNG_Init;
	_connectionTime = 3000;
	_one=1;
	_connect = TRUE;
	_potMsgLen = 0;
	_recvLen = 0;
	_recvOffset = 0;
	_counter = 0;
	SetSendDone(FALSE);
}

void MNG_ComHdlr::SetSendDone(bool toggle){
	_sendDone=toggle;
}

void MNG_ComHdlr::SetStateValue(MNG_internalState_t stateVal){
	_internalState=stateVal;
}
```

#### MNG_Global.hpp
```cpp
#ifndef  _MNGGLOBAL_HPP_
#define _MNGGLOBAL_HPP_

#include <mng_globalTYP.h>

    typedef struct {

		signed short NumSignals;

        /* BOOL diDriveParallelAtFront */
        BOOL diDriveParallelAtFront;
        /* BOOL diDriveParallelAtBack */
        BOOL diDriveParallelAtBack;
        /* BOOL diDriveCutAtFront */
        BOOL diDriveCutAtFront;
        /* BOOL diDriveCutAtBack */
        BOOL diDriveCutAtBack;

        } Saw_INPUTS_32BIT_FWRD;

    typedef struct {

		signed short NumSignals;

        /* BOOL doSawOn */
        BOOL doSawOn;
        /* LREAL aoTreeVelocity */
        REAL aoTreeVelocity;
        /* LREAL aoDriveParallelPosition */
        REAL aoDriveParallelPosition;
        /* LREAL aoDriveCutPosition */
        REAL aoDriveCutPosition;

        } Saw_OUTPUTS_32BIT_FWRD;

#endif
```

#### MNG_CpyOutToMsg.cpp
```cpp
#include "MNG_InternalTyp.hpp"

unsigned long int MNG_CpyOutToMsg(MNG_RawDatagram * pToServer, unsigned long int counter, Saw_OUTPUTS_32BIT_FWRD *pSimOutputs ) {

        unsigned long int DWordBuffer;

        pSimOutputs->NumSignals = 4;
        (pToServer->Header).ByteCount    = H_TO_NUDINT(20);
        (pToServer->Header).DatagramType = H_TO_NUDINT(MNG_Raw32BitImage);
        (pToServer->Header).SentTime = H_TO_NUDINT(0);  // Todo
        (pToServer->Header).Counter = H_TO_NUDINT(counter);
        pToServer->Payload[0] = H_TO_NUDINT(pSimOutputs->NumSignals);

    /* doSawOn : BOOL */
    if(pSimOutputs->doSawOn == 1) {
        pToServer->Payload[1] = 0xFFFFFFFF;   /*BOOL */
    } else {
        pToServer->Payload[1] = 0;
    }

    /* aoTreeVelocity : FLOAT64 */
    brsmemcpy((unsigned long int)&(DWordBuffer), (unsigned long int)&(pSimOutputs->aoTreeVelocity), 4);
    pToServer->Payload[2] = H_TO_NUDINT(DWordBuffer);

    /* aoDriveParallelPosition : FLOAT64 */
    brsmemcpy((unsigned long int)&(DWordBuffer), (unsigned long int)&(pSimOutputs->aoDriveParallelPosition), 4);
    pToServer->Payload[3] = H_TO_NUDINT(DWordBuffer);

    /* aoDriveCutPosition : FLOAT64 */
    brsmemcpy((unsigned long int)&(DWordBuffer), (unsigned long int)&(pSimOutputs->aoDriveCutPosition), 4);
    pToServer->Payload[4] = H_TO_NUDINT(DWordBuffer);

	return 0;
}
```

#### MNG_CpyMsgToInp.cpp
```cpp
#include "MNG_InternalTyp.hpp"

unsigned long int MNG_CpyMsgToInp(MNG_RawDatagram * pFromServer, Saw_INPUTS_32BIT_FWRD *pSimInputs) {

    MNG_DatagramType datagramType;
	unsigned long int DWordBuffer;
        unsigned long int byteCount;
	unsigned long int numSignalsInMessage;

	byteCount = N_TO_HUDINT((pFromServer->Header).ByteCount);
	datagramType = static_cast<MNG_DatagramType>(N_TO_HUDINT((pFromServer->Header).DatagramType));
	if (datagramType != MNG_Raw32BitImage) {
		return 0;
	}

    pSimInputs->NumSignals = 4;

    numSignalsInMessage = N_TO_HUDINT(pFromServer->Payload[0]);
        if ((static_cast<long int>(numSignalsInMessage) != pSimInputs->NumSignals) ||
	(byteCount != 4 + numSignalsInMessage * 4)) {
		return 0;
	}

    /* BOOL diDriveParallelAtFront */
    pSimInputs->diDriveParallelAtFront = (pFromServer->Payload[1] != 0);

    /* BOOL diDriveParallelAtBack */
    pSimInputs->diDriveParallelAtBack = (pFromServer->Payload[2] != 0);

    /* BOOL diDriveCutAtFront */
    pSimInputs->diDriveCutAtFront = (pFromServer->Payload[3] != 0);

    /* BOOL diDriveCutAtBack */
    pSimInputs->diDriveCutAtBack = (pFromServer->Payload[4] != 0);

return N_TO_HUDINT((pFromServer->Header).Counter); // return counter
}
```

### Program Logical/Libraries/Saw/Saw_P (ANSIC)

#### Main.cpp - Init, cyclic, exit code
```cpp
#include <bur/plctypes.h>

#include "../Saw_L/MNG_Global.hpp"
#include "../Saw_L/MNG_InternalTyp.hpp"
#include "../Saw_L/MNG_ComHdlr.hpp"

#include <MNG_PackageTyp.h>
#include <MNG_PackageVAR.h>
#include <TypesTYP.h>
#include <VariablesVAR.h>

unsigned long bur_heap_size = 0x4FFFF;

MNG_ComHdlr *pMNG_ComHdlr;

void _INIT ProgramInit(void)
{
    pMNG_ComHdlr = new MNG_ComHdlr(Saw_SimServerAddress, Saw_SimServerPort, Saw_SimSendCycleTime);
}

void _CYCLIC ProgramCyclic(void)
{

	connectionState = pMNG_ComHdlr->RunCommunication((void*)&Saw_SimInputs,(void*)&Saw_SimOutputs, &Saw_SimActive);

}
void _EXIT ProgramExit(void)
{
    delete pMNG_ComHdlr;
}
```

### MNG_Package.typ
```iecst
(*                                                                            *)
(* File generated by the B&R AS 4 control config generator                    *)
(*                                                                            *)
(*     Provider: machineering                                                 *)
(*  Application: industrialPhysics_2.4.master                                 *)
(* Architecture: Windows 64 Bit                                               *)
(*      Version: 2.4.11457.master                                             *)
(*        Build: 095f6f04a                                                    *)
(*         Date: 2020-10-12, Time: 08:55:42                                   *)
(*                                                                            *)

TYPE
Saw_INPUTS_32BIT : STRUCT

		NumSignals	: INT := 4;

        diDriveParallelAtFront : BOOL := 0;
        (* BOOL diDriveParallelAtFront *)
        diDriveParallelAtBack : BOOL := 0;
        (* BOOL diDriveParallelAtBack *)
        diDriveCutAtFront : BOOL := 0;
        (* BOOL diDriveCutAtFront *)
        diDriveCutAtBack : BOOL := 0;
        (* BOOL diDriveCutAtBack *)

	END_STRUCT;

Saw_OUTPUTS_32BIT : STRUCT

		NumSignals	: INT := 4;

        doSawOn : BOOL := 0;
        (* BOOL doSawOn *)
        aoTreeVelocity : REAL ;
        (* LREAL aoTreeVelocity *)
        aoDriveParallelPosition : REAL ;
        (* LREAL aoDriveParallelPosition *)
        aoDriveCutPosition : REAL ;
        (* LREAL aoDriveCutPosition *)

	END_STRUCT;

END_TYPE
```

### MNG_Package.var
```iecst
(*                                                                            *)
(* File generated by the B&R AS 4 control config generator                    *)
(*                                                                            *)
(*     Provider: machineering                                                 *)
(*  Application: industrialPhysics_2.4.master                                 *)
(* Architecture: Windows 64 Bit                                               *)
(*      Version: 2.4.11457.master                                             *)
(*        Build: 095f6f04a                                                    *)
(*         Date: 2020-10-12, Time: 08:55:42                                   *)
(*                                                                            *)
VAR
	Saw_SimInputs : Saw_INPUTS_32BIT := (0);
	Saw_SimOutputs : Saw_OUTPUTS_32BIT := (0);
	Saw_SimServerAddress : STRING[15] := '127.0.0.1';
	Saw_SimServerPort : UINT := 5000;
	Saw_SimSendCycleTime : TIME := T#5ms;
	Saw_SimActive : BOOL := FALSE;
END_VAR
```

### Program Logical/Main (IEC)

#### Types.typ
```iecst
TYPE
	StateMachineTyp :
		(
		INIT := 0,
		READY := 1,
		MANUAL := 2,
		AUTO := 3,
		ERROR := 4,
		WAIT_FOR_INIT
		);
END_TYPE
```

#### Variables.var
```iecst
VAR
	ResetErrors : BOOL;
	HMIman : BOOL;
	SwitchModeToMan : BOOL;
	StopAutoSequence : BOOL;
	StartAutoSequence : BOOL;
	diInitializeMachine : BOOL;
	SawRight : BOOL;
	SawOff : BOOL;
	SawBackward : BOOL;
	HMIauto : BOOL;
	ConveyorOff : BOOL;
	ConveyorOn : BOOL;
	SawOn : BOOL;
	SawForward : BOOL;
	SawLeft : BOOL;
	OperatingMode : INT;
	ParallelStep : REAL;
	PerpendicularStep : REAL;
	ConveyorSpeed : REAL;
	SMachine : StateMachineTyp;
	SwitchModeToAuto : BOOL;
END_VAR
```

#### Main.st
```iecst
PROGRAM _INIT
	ConveyorSpeed := 100;
	PerpendicularStep := 0.2;
	ParallelStep := 0.2;

	OperatingMode := 0;

	gStateSetter := 0;
	SMachine := WAIT_FOR_INIT;

	gInitProgressBarValue := 0;

	Saw_SimOutputs.doSawOn := gSawOn;

END_PROGRAM

PROGRAM _CYCLIC

	CASE SMachine OF
		INIT:
			gStateSetter := 1;

			IF gParallelSettings.doReadyToWork THEN
				gInitProgressBarValue := 60;

				IF gPerpendicularSettings.doReadyToWork THEN
					gInitProgressBarValue := 130;

					IF gConveyorSettings.doReadyToWork THEN
						gInitProgressBarValue := 200;

						SMachine := READY;
					END_IF;
				END_IF;
			END_IF;

		READY:
			gInitProgressBarValue := 255;

			IF HMIman THEN
	  			OperatingMode := 1;
			END_IF;

			IF HMIauto THEN
	  			OperatingMode := 2;
			END_IF;

			IF EDGEPOS(gOperatingPanel.diStart) THEN
				IF OperatingMode = 1 THEN
					gStateSetter := 2;
					SMachine := MANUAL;
				END_IF;

				IF OperatingMode = 2 THEN
					gStateSetter := 3;
	  				SMachine := AUTO;
				END_IF;
			END_IF;

		MANUAL:
			gConveyorSettings.aiSpeed := (ConveyorSpeed / 100);

			gParallelSettings.diLeft := SawLeft;
			gParallelSettings.diRight := SawRight;
			gParallelSettings.aiParallelStep := ParallelStep;

			gPerpendicularSettings.diForward := SawForward;
			gPerpendicularSettings.diBackward := SawBackward;
			gPerpendicularSettings.aiPerpendicularStep := PerpendicularStep;

			gOperatingPanel.SwitchModeToAuto := SwitchModeToAuto;

			IF SawOn THEN
				gSawOn := TRUE;
			END_IF;

			IF SawOff THEN
	  			gSawOn := FALSE;
			END_IF;

			IF ConveyorOn THEN
	  			gConveyorSettings.diRun := TRUE;
			END_IF;

			IF ConveyorOff THEN
				gConveyorSettings.diRun := FALSE;
			END_IF;

			IF gPerpendicularSettings.ReadyToChange AND gParallelSettings.ReadyToChange THEN
				IF SwitchModeToAuto THEN
					OperatingMode := 2;
					gStateSetter := 3;

					gParallelSettings.ReadyToChange := FALSE;
					gParallelSettings.AfterSwitchFlag := TRUE;
					gPerpendicularSettings.ReadyToChange := FALSE;
					gPerpendicularSettings.AfterSwitchFlag := TRUE;
					SwitchModeToAuto := FALSE;

					SMachine := AUTO;
				END_IF;
			END_IF;

		AUTO:
			gConveyorSettings.aiSpeed := (ConveyorSpeed / 100);

			gRecipeMenagement.Save1M := FALSE;
			gRecipeMenagement.Save2M := FALSE;
			gRecipeMenagement.Save3M := FALSE;

			gOperatingPanel.StartSequence := StartAutoSequence;
			gOperatingPanel.SwitchModeToMan := SwitchModeToMan;
			gOperatingPanel.StopSequence := StopAutoSequence;

			IF StartAutoSequence THEN
	  			gConveyorSettings.diRun := TRUE;
			END_IF;

			IF StopAutoSequence THEN
	  			gConveyorSettings.diRun := FALSE;
			END_IF;

			IF gOperatingPanel.SaveRecipe1M THEN
				gRecipe1M.AccTorqueLimit := gPerpendicularSettings.AccTorque;
				gRecipe1M.SawFeedRate := gPerpendicularSettings.FeedRate;
				gRecipe1M.WoodLogLength := gPerpendicularSettings.WoodLogLength;
				gRecipeMenagement.Save1M := TRUE;
			END_IF;

			IF gOperatingPanel.SaveRecipe2M THEN
				gRecipe2M.AccTorqueLimit := gPerpendicularSettings.AccTorque;
				gRecipe2M.SawFeedRate := gPerpendicularSettings.FeedRate;
				gRecipe2M.WoodLogLength := gPerpendicularSettings.WoodLogLength;
				gRecipeMenagement.Save2M := TRUE;
			END_IF;

			IF gOperatingPanel.SaveRecipe3M THEN
				gRecipe3M.AccTorqueLimit := gPerpendicularSettings.AccTorque;
				gRecipe3M.SawFeedRate := gPerpendicularSettings.FeedRate;
				gRecipe3M.WoodLogLength := gPerpendicularSettings.WoodLogLength;
				gRecipeMenagement.Save3M := TRUE;
			END_IF;

			IF gParallelSettings.ReadyToChange THEN
				IF StartAutoSequence THEN
					gParallelSettings.ReadyToChange := FALSE;
					gPerpendicularSettings.ReadyToChange := FALSE;
				END_IF;

				IF SwitchModeToMan THEN
					OperatingMode := 1;
					gStateSetter := 2;

					gParallelSettings.ReadyToChange := FALSE;
					gPerpendicularSettings.ReadyToChange := FALSE;
					SwitchModeToMan := FALSE;

					SMachine := MANUAL;
				END_IF;
			END_IF;

		ERROR:

		WAIT_FOR_INIT:
			IF EDGEPOS(diInitializeMachine) THEN
	  			SMachine := INIT;
			END_IF;

	END_CASE;

	Saw_SimOutputs.doSawOn := gSawOn;

	gResetErrors := ResetErrors;

END_PROGRAM

PROGRAM _EXIT
	(* Insert code here *)

END_PROGRAM
```

### Program Logical/ParallelAxis (IEC)

#### Types.typ
```iecst
TYPE
	WorkAutoProcessTyp :
		(
		START_POSITION := 0,
		READY := 1,
		CUT_SQ := 2,
		RETURN_SQ := 3,
		SWITCH_MODE := 4
		);
	InitProcessTyp :
		(
		INIT := 0,
		POWER := 1,
		HOME := 2,
		DONE := 3
		);
	WorkManProcessTyp :
		(
		WAIT := 0,
		RUN := 1,
		HOMEAGAIN := 2
		);
	MenagementTyp :
		(
		IDLE := 0,
		WARMUP := 1,
		WORK_M := 2,
		WORK_A := 3
		);
END_TYPE
```

#### Variables.var
```iecst
VAR
	StopSequence : BOOL;
	SequencePar : MpAxisCamSequencerParType;
	MpParallelPar : MpAxisBasicParType;
	MpAxisParallel : MpAxisBasic;
	InitMachine : InitProcessTyp;
	WorkManMachine : WorkManProcessTyp;
	MenageMachine : MenagementTyp;
	WorkAutoMachine : WorkAutoProcessTyp;
	SequencerParallel : MpAxisCamSequencer;
	McAcpCamPar : McAcpAxCamAutParType;
	RecipeLoadedStationaryFlag : BOOL;
END_VAR
```

#### Main.st
```iecst
PROGRAM _INIT
	MpParallelPar.Homing.Mode := 140;
	MpParallelPar.Velocity := 0.2;

	MpAxisParallel.Enable := TRUE;
	MpAxisParallel.MpLink := ADR(gParallelAxis);
	MpAxisParallel.Parameters := ADR(MpParallelPar);

	InitMachine := INIT;
	WorkManMachine := WAIT;
	WorkAutoMachine := START_POSITION;

	SequencePar.CamSequence.Data.DataAddress := ADR(McAcpCamPar);
	SequencePar.CamSequence.Data.DataSize := SIZEOF(McAcpCamPar);

	SequencePar.CamSequence.Set.Command := mcSET_UPDATE_FROM_ADR;
	SequencePar.CamSequence.Set.Mode := mcAXIS_CAM_SEQ_SET_ON_UPDATE;
	SequencePar.CamSequence.Get.Command := mcGET_PAR_ACTUAL;
	SequencePar.CamSequence.Get.GetOnEnable := TRUE;

END_PROGRAM

PROGRAM _CYCLIC
	MenageMachine := gStateSetter;

	CASE MenageMachine OF
		WARMUP:
			CASE InitMachine OF
				INIT:
					IF MpAxisParallel.Info.ReadyToPowerOn THEN
						InitMachine := POWER;
					END_IF;

				POWER:
					MpAxisParallel.Power := TRUE;

					IF MpAxisParallel.PowerOn THEN
						InitMachine := HOME;
					END_IF;

				HOME:
					MpAxisParallel.Home := TRUE;

					IF MpAxisParallel.IsHomed THEN
						MpAxisParallel.Home := FALSE;
						InitMachine := DONE;
					END_IF;

				DONE:
					gParallelSettings.doReadyToWork := TRUE;

			END_CASE;

		WORK_M:
			CASE WorkManMachine OF
				WAIT:
					MpAxisParallel.MoveAbsolute := FALSE;
					gParallelSettings.ReadyToChange := TRUE;

					IF EDGEPOS(gParallelSettings.diLeft) AND NOT(Saw_SimInputs.diDriveParallelAtFront) THEN
						MpParallelPar.Position := MpAxisParallel.Position + gParallelSettings.aiParallelStep;

						WorkManMachine := RUN;
					END_IF;

					IF EDGEPOS(gParallelSettings.diRight) AND NOT(Saw_SimInputs.diDriveParallelAtBack) THEN
						MpParallelPar.Position := MpAxisParallel.Position - gParallelSettings.aiParallelStep;

						WorkManMachine := RUN;
					END_IF;

					IF EDGEPOS(gOperatingPanel.diHomeParallel) THEN
						WorkManMachine := HOMEAGAIN;
					END_IF;

				RUN:
					MpAxisParallel.MoveAbsolute := TRUE;
					gParallelSettings.ReadyToChange := FALSE;

					IF MpAxisParallel.MoveDone THEN
						WorkManMachine := WAIT;
					END_IF;

					IF EDGENEG(MpAxisParallel.Error) THEN
	  					WorkManMachine := WAIT;
					END_IF;

				HOMEAGAIN:
					MpAxisParallel.Home := TRUE;
					gParallelSettings.ReadyToChange := FALSE;

					IF EDGEPOS(MpAxisParallel.IsHomed) THEN
						MpAxisParallel.Home := FALSE;
						WorkManMachine := WAIT;
					END_IF;

			END_CASE;

		WORK_A:
			CASE WorkAutoMachine OF
				START_POSITION:

					MpParallelPar.Position := -0.25;
					MpAxisParallel.MoveAbsolute := TRUE;

					IF MpAxisParallel.MoveDone THEN
						MpAxisParallel.MoveAbsolute := FALSE;
						WorkAutoMachine := READY;

					END_IF;

				READY:
					IF gParallelSettings.AfterSwitchFlag THEN
						gParallelSettings.AfterSwitchFlag := FALSE;
						WorkAutoMachine := START_POSITION;
					END_IF;

					gParallelSettings.AutoReady := TRUE;

					IF gOperatingPanel.StartSequence THEN
						WorkAutoMachine := CUT_SQ;

					END_IF;

					IF gOperatingPanel.LoadRecipe1M THEN
						gParallelSettings.AutoReady := FALSE;
						RecipeLoadedStationaryFlag := TRUE;

						WorkAutoMachine := LOAD_1M;
					END_IF;

					IF gOperatingPanel.LoadRecipe2M THEN
						gParallelSettings.AutoReady := FALSE;
						RecipeLoadedStationaryFlag := TRUE;

						WorkAutoMachine := LOAD_2M;
					END_IF;

					IF gOperatingPanel.LoadRecipe3M THEN
						gParallelSettings.AutoReady := FALSE;
						RecipeLoadedStationaryFlag := TRUE;

						WorkAutoMachine := LOAD_3M;
					END_IF;

				CUT_SQ:
					SequencerParallel.StartSequence := TRUE;

					IF SequencerParallel.InCam THEN
	  					WorkAutoMachine := RETURN_SQ;
					END_IF;

				RETURN_SQ:
					IF gOperatingPanel.StopSequence THEN
						StopSequence := TRUE;
					END_IF;

					SequencerParallel.Signal1 := StopSequence;

					IF StopSequence THEN
						StopSequence := FALSE;
						SequencerParallel.StartSequence := FALSE;

						WorkAutoMachine := SWITCH_MODE;
					END_IF;

					IF gOperatingPanel.LoadRecipe1M THEN
	  					WorkAutoMachine := LOAD_1M;
					END_IF;

					IF gOperatingPanel.LoadRecipe2M THEN
						WorkAutoMachine := LOAD_2M;
					END_IF;

					IF gOperatingPanel.LoadRecipe3M THEN
	  					WorkAutoMachine := LOAD_3M;
					END_IF;

				SWITCH_MODE:
					IF gPerpendicularSettings.ReadyToChange THEN
						MpParallelPar.Position := -0.25;
						MpAxisParallel.MoveAbsolute := TRUE;

						IF MpAxisParallel.MoveDone THEN
							MpAxisParallel.MoveAbsolute := FALSE;
							gParallelSettings.ReadyToChange := TRUE;

							WorkAutoMachine := READY;
						END_IF;
					END_IF;

				LOAD_1M:
					McAcpCamPar.State[1].MasterFactor := 300;
					McAcpCamPar.State[1].SlaveFactor := 300;

					McAcpCamPar.State[1].CompensationMode := mcCOMP_BETWEEN_CAMS_DIRECT;
					McAcpCamPar.State[1].CompensationParameters.MasterCompDistance := 0.2;
					McAcpCamPar.State[1].CompensationParameters.SlaveCompDistance := 0.2;

					McAcpCamPar.State[2].MasterFactor := 300;
					McAcpCamPar.State[2].SlaveFactor := -300;

					McAcpCamPar.State[2].CompensationMode := mcCOMP_BETWEEN_CAMS_DIRECT;
					McAcpCamPar.State[2].CompensationParameters.MasterCompDistance := 0.2;
					McAcpCamPar.State[2].CompensationParameters.SlaveCompDistance := -0.2;

					SequencerParallel.Update := TRUE;

					IF SequencerParallel.UpdateDone THEN
						SequencerParallel.Update := FALSE;

						IF RecipeLoadedStationaryFlag THEN
							RecipeLoadedStationaryFlag := FALSE;
							WorkAutoMachine := READY;
						ELSE
							WorkAutoMachine := RETURN_SQ;
						END_IF;

					END_IF;

				LOAD_2M:
					McAcpCamPar.State[1].MasterFactor := 300;
					McAcpCamPar.State[1].SlaveFactor := 300;

					McAcpCamPar.State[1].CompensationMode := mcCOMP_BETWEEN_CAMS_DIRECT;
					McAcpCamPar.State[1].CompensationParameters.MasterCompDistance := 0.2;
					McAcpCamPar.State[1].CompensationParameters.SlaveCompDistance := 0.2;

					McAcpCamPar.State[2].MasterFactor := 1200;
					McAcpCamPar.State[2].SlaveFactor := -300;

					McAcpCamPar.State[2].CompensationMode := mcCOMP_BETWEEN_CAMS_DIRECT;
					McAcpCamPar.State[2].CompensationParameters.MasterCompDistance := 0.3;
					McAcpCamPar.State[2].CompensationParameters.SlaveCompDistance := -0.2;

					SequencerParallel.Update := TRUE;

					IF SequencerParallel.UpdateDone THEN
						SequencerParallel.Update := FALSE;

						IF RecipeLoadedStationaryFlag THEN
							RecipeLoadedStationaryFlag := FALSE;
							WorkAutoMachine := READY;
						ELSE
							WorkAutoMachine := RETURN_SQ;
						END_IF;
					END_IF;

				LOAD_3M:
					McAcpCamPar.State[1].MasterFactor := 300;
					McAcpCamPar.State[1].SlaveFactor := 300;

					McAcpCamPar.State[1].CompensationMode := mcCOMP_BETWEEN_CAMS_DIRECT;
					McAcpCamPar.State[1].CompensationParameters.MasterCompDistance := 0.2;
					McAcpCamPar.State[1].CompensationParameters.SlaveCompDistance := 0.2;

					McAcpCamPar.State[2].MasterFactor := 2200;
					McAcpCamPar.State[2].SlaveFactor := -300;

					McAcpCamPar.State[2].CompensationMode := mcCOMP_BETWEEN_CAMS_DIRECT;
					McAcpCamPar.State[2].CompensationParameters.MasterCompDistance := 0.3;
					McAcpCamPar.State[2].CompensationParameters.SlaveCompDistance := -0.2;

					SequencerParallel.Update := TRUE;

					IF SequencerParallel.UpdateDone THEN
						SequencerParallel.Update := FALSE;

						IF RecipeLoadedStationaryFlag THEN
							RecipeLoadedStationaryFlag := FALSE;
							WorkAutoMachine := READY;
						ELSE
							WorkAutoMachine := RETURN_SQ;
						END_IF;
					END_IF;
			END_CASE;

		IDLE:

	END_CASE;

	SequencerParallel(MpLink := ADR(gParallelAxis), Enable := TRUE, Parameters := ADR(SequencePar), MpLinkMaster := ADR(gConveyorAxis));
	//MpAxisCamSequencer_0(MpLink := , Enable := , ErrorReset := , Parameters := , Update := , MpLinkMaster := , Signal1 := , Signal2 := , Signal3 := , Signal4 := , StartSequence := , Continue := , EndSequence := , GetSequence := , ParLock := , OffsetShift := , PhaseShift := , CamPrepare := , Recovery := );

	MpAxisParallel.ErrorReset := gResetErrors;

	Saw_SimOutputs.aoDriveParallelPosition := LREAL_TO_REAL(MpAxisParallel.Position);
	MpAxisParallel();

END_PROGRAM

PROGRAM _EXIT
	(* Insert code here *)

END_PROGRAM
```

### Program Logical/PerpendicularAxis (IEC)

#### Types.typ
```iecst
TYPE
	WorkAutoProcessTyp :
		(
		START_POSITION := 0,
		READY := 1,
		CUT_SQ := 2,
		RETURN_SQ := 3,
		SWITCH_MODE := 4,
		LOAD_1M := 5,
		LOAD_2M := 6,
		LOAD_3M := 7
		);
	InitProcessTyp :
		(
		INIT := 0,
		POWER := 1,
		HOME := 2,
		DONE := 3
		);
	WorkManProcessTyp :
		(
		WAIT := 0,
		RUN := 1,
		HOMEAGAIN := 2
		);
	MenagementTyp :
		(
		IDLE := 0,
		WARMUP := 1,
		WORK_M := 2,
		WORK_A := 3
		);
END_TYPE
```

#### Variables.var
```iecst
VAR
	RecipeLoadedStationaryFlag : BOOL;
	StopSequence : BOOL;
	InitMachine : InitProcessTyp;
	MenageMachine : MenagementTyp;
	MpAxisPerpendicular : MpAxisBasic;
	MpPerpendicularPar : MpAxisBasicParType;
	SequencerPerpendicular : MpAxisCamSequencer;
	SequencePar : MpAxisCamSequencerParType;
	WorkAutoMachine : WorkAutoProcessTyp;
	WorkManMachine : WorkManProcessTyp;
	McAcpCamPar : McAcpAxCamAutParType;
END_VAR
```

#### Main.st
```iecst
PROGRAM _INIT
	MpPerpendicularPar.Homing.Mode := 140;
	MpPerpendicularPar.Velocity := 0.2;

	MpAxisPerpendicular.Enable := TRUE;
	MpAxisPerpendicular.MpLink := ADR(gPerpendicularAxis);
	MpAxisPerpendicular.Parameters := ADR(MpPerpendicularPar);

	InitMachine := INIT;
	WorkManMachine := WAIT;
	WorkAutoMachine := START_POSITION;

	SequencePar.CamSequence.Data.DataAddress := ADR(McAcpCamPar);
	SequencePar.CamSequence.Data.DataSize := SIZEOF(McAcpCamPar);

	SequencePar.CamSequence.Set.Command := mcSET_UPDATE_FROM_ADR;
	SequencePar.CamSequence.Set.Mode := mcAXIS_CAM_SEQ_SET_ON_UPDATE;
	SequencePar.CamSequence.Get.Command := mcGET_PAR_ACTUAL;
	SequencePar.CamSequence.Get.GetOnEnable := TRUE;

END_PROGRAM

PROGRAM _CYCLIC
	MenageMachine := gStateSetter;

	CASE MenageMachine OF
		WARMUP:
			CASE InitMachine OF
				INIT:
					IF MpAxisPerpendicular.Info.ReadyToPowerOn THEN
						InitMachine := POWER;
					END_IF;

				POWER:
					MpAxisPerpendicular.Power := TRUE;

					IF MpAxisPerpendicular.PowerOn THEN
						InitMachine := HOME;
					END_IF;

				HOME:
					MpAxisPerpendicular.Home := TRUE;

					IF MpAxisPerpendicular.IsHomed THEN
						MpAxisPerpendicular.Home := FALSE;
						InitMachine := DONE;
					END_IF;

				DONE:
					gPerpendicularSettings.doReadyToWork := TRUE;

			END_CASE;

		WORK_M:
			CASE WorkManMachine OF
				WAIT:
					MpAxisPerpendicular.MoveAbsolute := FALSE;
					gPerpendicularSettings.ReadyToChange := TRUE;

					IF EDGEPOS(gPerpendicularSettings.diForward) AND NOT(Saw_SimInputs.diDriveCutAtFront) THEN
						MpPerpendicularPar.Position := MpAxisPerpendicular.Position + gPerpendicularSettings.aiPerpendicularStep;

						WorkManMachine := RUN;
					END_IF;

					IF EDGEPOS(gPerpendicularSettings.diBackward) AND NOT(Saw_SimInputs.diDriveCutAtBack) THEN
						MpPerpendicularPar.Position := MpAxisPerpendicular.Position - gPerpendicularSettings.aiPerpendicularStep;

						WorkManMachine := RUN;
					END_IF;

					IF EDGEPOS(gOperatingPanel.diHomePerpendicular) THEN
						WorkManMachine := HOMEAGAIN;
					END_IF;

				RUN:
					MpAxisPerpendicular.MoveAbsolute := TRUE;
					gPerpendicularSettings.ReadyToChange := FALSE;

					IF MpAxisPerpendicular.MoveDone THEN
						WorkManMachine := WAIT;
					END_IF;

					IF EDGENEG(MpAxisPerpendicular.Error) THEN
						WorkManMachine := WAIT;
					END_IF;

				HOMEAGAIN:
					MpAxisPerpendicular.Home := TRUE;
					gPerpendicularSettings.ReadyToChange := FALSE;

					IF EDGEPOS(MpAxisPerpendicular.IsHomed) THEN
						MpAxisPerpendicular.Home := FALSE;
						WorkManMachine := WAIT;
					END_IF;

			END_CASE;

		WORK_A:
			CASE WorkAutoMachine OF
				START_POSITION:
					MpPerpendicularPar.Position := 0.4;
					MpAxisPerpendicular.MoveAbsolute := TRUE;

					IF MpAxisPerpendicular.MoveDone THEN
						MpAxisPerpendicular.MoveAbsolute := FALSE;
						WorkAutoMachine := READY;

					END_IF;

				READY:
					IF gPerpendicularSettings.AfterSwitchFlag THEN
						gPerpendicularSettings.AfterSwitchFlag := FALSE;
						WorkAutoMachine := START_POSITION;
					END_IF;

					gPerpendicularSettings.AutoReady := TRUE;

					IF gOperatingPanel.StartSequence THEN
						gSawOn := TRUE;
						WorkAutoMachine := CUT_SQ;

					END_IF;

					IF gOperatingPanel.LoadRecipe1M THEN
						RecipeLoadedStationaryFlag := TRUE;
						gPerpendicularSettings.AutoReady := FALSE;

						WorkAutoMachine := LOAD_1M;
					END_IF;

					IF gOperatingPanel.LoadRecipe2M THEN
						RecipeLoadedStationaryFlag := TRUE;
						gPerpendicularSettings.AutoReady := FALSE;

						WorkAutoMachine := LOAD_2M;
					END_IF;

					IF gOperatingPanel.LoadRecipe3M THEN
						RecipeLoadedStationaryFlag := TRUE;
						gPerpendicularSettings.AutoReady := FALSE;

						WorkAutoMachine := LOAD_3M;
					END_IF;

				CUT_SQ:
					SequencerPerpendicular.StartSequence := TRUE;

					IF SequencerPerpendicular.InCam THEN
	  					WorkAutoMachine := RETURN_SQ;
					END_IF;

				RETURN_SQ:
					SequencerPerpendicular.Continue := FALSE;

					IF gOperatingPanel.StopSequence THEN
	  					StopSequence := TRUE;
					END_IF;

					SequencerPerpendicular.Signal1 := StopSequence;

					IF StopSequence THEN
						StopSequence := FALSE;
						SequencerPerpendicular.StartSequence := FALSE;

						WorkAutoMachine := SWITCH_MODE;
					END_IF;

					IF gOperatingPanel.LoadRecipe1M THEN
						WorkAutoMachine := LOAD_1M;
					END_IF;

					IF gOperatingPanel.LoadRecipe2M THEN
						WorkAutoMachine := LOAD_2M;
					END_IF;

					IF gOperatingPanel.LoadRecipe3M THEN
						WorkAutoMachine := LOAD_3M;
					END_IF;

				SWITCH_MODE:
					MpPerpendicularPar.Position := 0.4;
					MpAxisPerpendicular.MoveAbsolute := TRUE;

					IF MpAxisPerpendicular.MoveDone THEN
						MpAxisPerpendicular.MoveAbsolute := FALSE;
						gPerpendicularSettings.ReadyToChange := TRUE;
						gSawOn := FALSE;

						WorkAutoMachine := READY;
					END_IF;

				LOAD_1M:
					gRecipeMenagement.Load1M := TRUE;
					gPerpendicularSettings.AccTorque := gRecipe1M.AccTorqueLimit;
					gPerpendicularSettings.FeedRate := gRecipe1M.SawFeedRate;
					gPerpendicularSettings.WoodLogLength := gRecipe1M.WoodLogLength;

					McAcpCamPar.State[1].MasterFactor := 125;
					McAcpCamPar.State[1].SlaveFactor := 300;
					McAcpCamPar.State[1].CompensationMode := mcCOMP_BETWEEN_CAMS_DIRECT;
					McAcpCamPar.State[1].CompensationParameters.MasterCompDistance := 0.125;
					McAcpCamPar.State[1].CompensationParameters.SlaveCompDistance := 0.2;

					McAcpCamPar.State[2].MasterFactor := 125;
					McAcpCamPar.State[2].SlaveFactor := -300;
					McAcpCamPar.State[2].CompensationMode := mcCOMP_BETWEEN_CAMS_DIRECT;
					McAcpCamPar.State[2].CompensationParameters.MasterCompDistance := 0.125;
					McAcpCamPar.State[2].CompensationParameters.SlaveCompDistance := -0.2;

					McAcpCamPar.State[3].MasterFactor := 500;
					McAcpCamPar.State[3].SlaveFactor := 0;
					McAcpCamPar.State[3].CompensationMode := mcCOMP_OFF;

					SequencerPerpendicular.Update := TRUE;

					IF SequencerPerpendicular.UpdateDone THEN
						SequencerPerpendicular.Update := FALSE;
						gRecipeMenagement.Load1M := FALSE;

						IF RecipeLoadedStationaryFlag THEN
							RecipeLoadedStationaryFlag := FALSE;
							WorkAutoMachine := READY;
						ELSE
							WorkAutoMachine := RETURN_SQ;
						END_IF;
					END_IF;

				LOAD_2M:
					gRecipeMenagement.Load2M := TRUE;
					gPerpendicularSettings.AccTorque := gRecipe2M.AccTorqueLimit;
					gPerpendicularSettings.FeedRate := gRecipe2M.SawFeedRate;
					gPerpendicularSettings.WoodLogLength := gRecipe2M.WoodLogLength;

					McAcpCamPar.State[1].MasterFactor := 125;
					McAcpCamPar.State[1].SlaveFactor := 300;
					McAcpCamPar.State[1].CompensationParameters.MasterCompDistance := 0.125;
					McAcpCamPar.State[1].CompensationParameters.SlaveCompDistance := 0.2;

					McAcpCamPar.State[2].MasterFactor := 125;
					McAcpCamPar.State[2].SlaveFactor := -300;
					McAcpCamPar.State[2].CompensationParameters.MasterCompDistance := 0.125;
					McAcpCamPar.State[2].CompensationParameters.SlaveCompDistance := -0.2;

					McAcpCamPar.State[3].MasterFactor := 1500;
					McAcpCamPar.State[3].SlaveFactor := 0;
					McAcpCamPar.State[3].CompensationMode := mcCOMP_OFF;

					SequencerPerpendicular.Update := TRUE;

					IF SequencerPerpendicular.UpdateDone THEN
						SequencerPerpendicular.Update := FALSE;
						gRecipeMenagement.Load2M := FALSE;

						IF RecipeLoadedStationaryFlag THEN
							RecipeLoadedStationaryFlag := FALSE;
							WorkAutoMachine := READY;
						ELSE
							WorkAutoMachine := RETURN_SQ;
						END_IF;
					END_IF;

				LOAD_3M:
					gRecipeMenagement.Load3M := TRUE;
					gPerpendicularSettings.AccTorque := gRecipe3M.AccTorqueLimit;
					gPerpendicularSettings.FeedRate := gRecipe3M.SawFeedRate;
					gPerpendicularSettings.WoodLogLength := gRecipe3M.WoodLogLength;

					McAcpCamPar.State[1].MasterFactor := 125;
					McAcpCamPar.State[1].SlaveFactor := 200;
					McAcpCamPar.State[1].CompensationParameters.MasterCompDistance := 0.125;
					McAcpCamPar.State[1].CompensationParameters.SlaveCompDistance := 0.3;

					McAcpCamPar.State[2].MasterFactor := 125;
					McAcpCamPar.State[2].SlaveFactor := -200;
					McAcpCamPar.State[2].CompensationParameters.MasterCompDistance := 0.125;
					McAcpCamPar.State[2].CompensationParameters.SlaveCompDistance := -0.3;

					McAcpCamPar.State[3].MasterFactor := 2500;
					McAcpCamPar.State[3].SlaveFactor := 0;
					McAcpCamPar.State[3].CompensationMode := mcCOMP_OFF;

					SequencerPerpendicular.Update := TRUE;

					IF SequencerPerpendicular.UpdateDone THEN
						SequencerPerpendicular.Update := FALSE;
						gRecipeMenagement.Load3M := FALSE;

						IF RecipeLoadedStationaryFlag THEN
							RecipeLoadedStationaryFlag := FALSE;
							WorkAutoMachine := READY;
						ELSE
							WorkAutoMachine := RETURN_SQ;
						END_IF;
					END_IF;

			END_CASE;

		IDLE:

	END_CASE;

	SequencerPerpendicular(MpLink := ADR(gPerpendicularAxis), Enable := TRUE, Parameters := ADR(SequencePar), MpLinkMaster := ADR(gConveyorAxis));

	MpAxisPerpendicular.ErrorReset := gResetErrors;

	Saw_SimOutputs.aoDriveCutPosition := LREAL_TO_REAL(MpAxisPerpendicular.Position);
	MpAxisPerpendicular();

END_PROGRAM

PROGRAM _EXIT
	(* Insert code here *)

END_PROGRAM
```

### Program Logical/ConveyorAxis (IEC)

#### Types.typ
```iecst
TYPE
	InitProcessTyp :
		(
		INIT := 0,
		POWER := 1,
		HOME := 2,
		DONE := 3
		);
	WorkProcessTyp :
		(
		WAIT := 0,
		RUN := 1,
		UPDATE
		);
	MenagementTyp :
		(
		IDLE := 0,
		WARMUP := 1,
		WORK_M := 2,
		WORK_A := 3
		);
END_TYPE
```

#### Variables.var
```iecst
VAR
	WorkAutoMachine : WorkProcessTyp;
	MpConveyorPar : MpAxisBasicParType;
	MpAxisConveyor : MpAxisBasic;
	InitMachine : InitProcessTyp;
	WorkManMachine : WorkProcessTyp;
	MenageMachine : MenagementTyp;
END_VAR
```

#### Main.st
```iecst
PROGRAM _INIT
	MpAxisConveyor.Enable := TRUE;
	MpAxisConveyor.MpLink := ADR(gConveyorAxis);
	MpAxisConveyor.Parameters := ADR(MpConveyorPar);

	InitMachine := INIT;
	WorkManMachine := WAIT;
	WorkAutoMachine := WAIT;

END_PROGRAM

PROGRAM _CYCLIC
	MpAxisConveyor();
	MenageMachine := gStateSetter;

	CASE MenageMachine OF
		IDLE:

		WARMUP:
			CASE InitMachine OF
				INIT:
					IF MpAxisConveyor.Info.ReadyToPowerOn THEN
						InitMachine := POWER;
					END_IF;

				POWER:
					MpAxisConveyor.Power := TRUE;

					IF MpAxisConveyor.PowerOn THEN
						InitMachine := HOME;
					END_IF;

				HOME:
					MpAxisConveyor.Home := TRUE;

					IF MpAxisConveyor.IsHomed THEN
						InitMachine := DONE;
					END_IF;

				DONE:
					gConveyorSettings.doReadyToWork := TRUE;

			END_CASE;

		WORK_M:
			CASE WorkManMachine OF
				WAIT:
					MpAxisConveyor.MoveVelocity := FALSE;

					IF gConveyorSettings.diRun THEN
	  					WorkManMachine := RUN;
					END_IF;

				RUN:
					MpAxisConveyor.MoveVelocity := TRUE;

					IF NOT(MpConveyorPar.Velocity = gConveyorSettings.aiSpeed) THEN
						WorkManMachine := UPDATE;
					END_IF;

					IF NOT(gConveyorSettings.diRun) THEN
						WorkManMachine := WAIT;
					END_IF;

				UPDATE:
					MpConveyorPar.Velocity := gConveyorSettings.aiSpeed;
					MpAxisConveyor.Update := TRUE;

					IF MpAxisConveyor.UpdateDone THEN
						MpAxisConveyor.Update := FALSE;
	  					WorkManMachine := RUN;
					END_IF;
			END_CASE;

		WORK_A:
			CASE WorkAutoMachine OF
				WAIT:
					MpConveyorPar.Velocity := gConveyorSettings.aiSpeed;
					MpAxisConveyor.MoveVelocity := FALSE;

					IF gConveyorSettings.diRun THEN
						WorkAutoMachine := RUN;
					END_IF;
				RUN:
					MpAxisConveyor.MoveVelocity := TRUE;

					IF NOT(MpConveyorPar.Velocity = gConveyorSettings.aiSpeed) THEN
						WorkAutoMachine := UPDATE;
					END_IF;

					IF NOT(gConveyorSettings.diRun) THEN
						MpAxisConveyor.MoveVelocity := FALSE;
						WorkAutoMachine := WAIT;
					END_IF;

				UPDATE:
					MpConveyorPar.Velocity := gConveyorSettings.aiSpeed;
					MpAxisConveyor.Update := TRUE;

					IF MpAxisConveyor.UpdateDone THEN
						MpAxisConveyor.Update := FALSE;
						WorkAutoMachine := RUN;
					END_IF;

			END_CASE;

	END_CASE;

	Saw_SimOutputs.aoTreeVelocity := MpAxisConveyor.Velocity;

	MpAxisConveyor.ErrorReset := gResetErrors;

END_PROGRAM

PROGRAM _EXIT
	(* Insert code here *)

END_PROGRAM
```

### Program Logical/Alarm (IEC)

#### Variables.var
```iecst
VAR
	MpAlarmXListUI_0 : MpAlarmXListUI;
	MpAlarmXCore_0 : MpAlarmXCore;
	MpAlarmXHistory_0 : MpAlarmXHistory;
END_VAR
```

#### Main.st
```iecst
PROGRAM _INIT
	(* Insert code here *)
	MpAlarmXCore_0.Enable := TRUE;
	MpAlarmXCore_0.MpLink := ADR(gAlarmXCore);

	MpAlarmXListUI_0.Enable := TRUE;
	MpAlarmXListUI_0.MpLink := ADR(gAlarmXCore);

	MpAlarmXHistory_0.Enable := TRUE;
	MpAlarmXHistory_0.MpLink := ADR(gAlarmXHistory);

END_PROGRAM

PROGRAM _CYCLIC
	(* Insert code here *)
	MpAlarmXCore_0();
	MpAlarmXListUI_0();

	MpAlarmXHistory_0();

END_PROGRAM

PROGRAM _EXIT
	(* Insert code here *)

END_PROGRAM
```

### Program Logical/Recipe (IEC)

#### Variables.var
```iecst
VAR
	MpRecipeXml_0 : MpRecipeXml;
	MpRecipeRegPar_0 : MpRecipeRegPar;
	MpRecipeXml_1 : MpRecipeXml;
	MpRecipeRegPar_1 : MpRecipeRegPar;
	MpRecipeXml_2 : MpRecipeXml;
	MpRecipeRegPar_2 : MpRecipeRegPar;
END_VAR
```

#### Main.st
```iecst
PROGRAM _INIT
	gRecipe1M.SawFeedRate := gRecipe1M.SawFeedRate;
	gRecipe2M.SawFeedRate := gRecipe2M.SawFeedRate;
	gRecipe3M.SawFeedRate := gRecipe3M.SawFeedRate;

	gPerpendicularSettings.AutoReady := gPerpendicularSettings.AutoReady;

	MpRecipeXml_0(MpLink := ADR(gRecipeXml), Enable := TRUE, DeviceName := ADR('USER'), FileName := ADR('Recipe1m'));
	MpRecipeRegPar_0(MpLink := ADR(gRecipeXml), Enable := TRUE, PVName := ADR('gRecipe1M'));

	MpRecipeXml_1(MpLink := ADR(gRecipeXml_1), Enable := TRUE, DeviceName := ADR('USER'), FileName := ADR('Recipe2m'));
	MpRecipeRegPar_1(MpLink := ADR(gRecipeXml_1), Enable := TRUE, PVName := ADR('gRecipe2M'));

	MpRecipeXml_2(MpLink := ADR(gRecipeXml_2), Enable := TRUE, DeviceName := ADR('USER'), FileName := ADR('Recipe3m'));
	MpRecipeRegPar_2(MpLink := ADR(gRecipeXml_2), Enable := TRUE, PVName := ADR('gRecipe3M'));

END_PROGRAM

PROGRAM _CYCLIC
	MpRecipeXml_0.Save := gRecipeMenagement.Save1M;
	MpRecipeXml_0.Load := gRecipeMenagement.Load1M;

	MpRecipeXml_1.Save := gRecipeMenagement.Save2M;
	MpRecipeXml_1.Load := gRecipeMenagement.Load2M;

	MpRecipeXml_2.Save := gRecipeMenagement.Save3M;
	MpRecipeXml_2.Load := gRecipeMenagement.Load3M;

	MpRecipeXml_0();
	MpRecipeRegPar_0();

	MpRecipeXml_1();
	MpRecipeRegPar_1();

	MpRecipeXml_2();
	MpRecipeRegPar_2();

END_PROGRAM

PROGRAM _EXIT
	(* Insert code here *)

END_PROGRAM
```

- Visualisation Logical/mappView (not shown)

### Program Logical/OsProstopadla

#### Types.typ
```iecst
TYPE
	StateMachineTyp :
		(
		INIT := 0,
		POWER := 1,
		HOME := 2,
		WAIT := 3,
		RUNB := 4,
		RUNF := 5
	);
END_TYPE
```

#### Variables.var
```iecst
VAR
	MpPerpendicularPar : MpAxisBasicParType;
	MpAxisPerpendicular : MpAxisBasic;
	SMachine : StateMachineTyp;
END_VAR
```

#### Main.st
```iecst
PROGRAM _INIT
	MpAxisPerpendicular.Enable := TRUE;
	MpAxisPerpendicular.MpLink := ADR(gPerpendicularAxis);
	MpAxisPerpendicular.Parameters := ADR(MpPerpendicularPar);

	SMachine := INIT;

END_PROGRAM

PROGRAM _CYCLIC

	MpAxisPerpendicular();

	CASE SMachine OF
		INIT:
			MpAxisPerpendicular.Power := FALSE;
			MpAxisPerpendicular.Home := FALSE;

			IF EDGEPOS(gPerpendicularAxisSettings.diRunAxis) AND MpAxisPerpendicular.Info.ReadyToPowerOn THEN
	  			SMachine := POWER;
			END_IF;

		POWER:
			MpAxisPerpendicular.Power := TRUE;

			IF MpAxisPerpendicular.PowerOn THEN
	  			SMachine := HOME;
			END_IF;

		HOME:
			IF NOT(MpAxisPerpendicular.IsHomed) THEN
				MpAxisPerpendicular.Home := TRUE;
			END_IF;

			IF MpAxisPerpendicular.IsHomed THEN
				SMachine := WAIT;
			END_IF;

		WAIT:
			MpAxisPerpendicular.MoveAbsolute := FALSE;

			IF EDGEPOS(gPerpendicularAxisSettings.diBackward) AND NOT(Saw_SimInputs.diDriveCutAtBack) THEN
				MpPerpendicularPar.Position := MpAxisPerpendicular.Position - gPerpendicularAxisSettings.aiPerpendicularStep;
				Saw_SimOutputs.aoDriveCutPosition := Saw_SimOutputs.aoDriveCutPosition - gPerpendicularAxisSettings.aiPerpendicularStep;

				SMachine := RUNB;
			END_IF;

			IF EDGEPOS(gPerpendicularAxisSettings.diForward) AND NOT(Saw_SimInputs.diDriveCutAtFront) THEN
				MpPerpendicularPar.Position := MpAxisPerpendicular.Position + gPerpendicularAxisSettings.aiPerpendicularStep;
				Saw_SimOutputs.aoDriveCutPosition := Saw_SimOutputs.aoDriveCutPosition + gPerpendicularAxisSettings.aiPerpendicularStep;

				SMachine := RUNF;
			END_IF;

			IF NOT(gPerpendicularAxisSettings.diRunAxis) THEN
				SMachine := INIT;
			END_IF;

		RUNB:
			MpAxisPerpendicular.MoveAbsolute := TRUE;

			IF MpAxisPerpendicular.MoveDone THEN
				SMachine := WAIT;
			END_IF;

		RUNF:
			MpAxisPerpendicular.MoveAbsolute := TRUE;

			IF MpAxisPerpendicular.MoveDone THEN
				SMachine := WAIT;
			END_IF;

	END_CASE;

END_PROGRAM

PROGRAM _EXIT
	(* Insert code here *)

END_PROGRAM
```

### Program Logical/OsRownolegla

#### Types.typ
```iecst
TYPE
	StateMachineTyp :
		(
		INIT := 0,
		POWER := 1,
		HOME := 2,
		WAIT := 3,
		RUNL := 4,
		RUNR := 5
		);
END_TYPE
```

#### Variables.var
```iecst
VAR
	MpParallelPar : MpAxisBasicParType;
	MpAxisParallel : MpAxisBasic;
	SMachine : StateMachineTyp;
END_VAR
```

#### Main.st
```iecst
PROGRAM _INIT
	MpAxisParallel.Enable := TRUE;
	MpAxisParallel.MpLink := ADR(gParallelAxis);
	MpAxisParallel.Parameters := ADR(MpParallelPar);

	SMachine := INIT;

END_PROGRAM

PROGRAM _CYCLIC
	MpAxisParallel();

	CASE SMachine OF
		INIT:
			MpAxisParallel.Power := FALSE;
			MpAxisParallel.Home := FALSE;

			IF EDGEPOS(gParallelAxisSettings.diRunAxis) AND MpAxisParallel.Info.ReadyToPowerOn THEN
	  			SMachine := POWER;
			END_IF;

		POWER:
			MpAxisParallel.Power := TRUE;

			IF MpAxisParallel.PowerOn THEN
	  			SMachine := HOME;
			END_IF;

		HOME:
			IF NOT(MpAxisParallel.IsHomed) THEN
				MpAxisParallel.Home := TRUE;
			END_IF;

			IF MpAxisParallel.IsHomed THEN
				SMachine := WAIT;
			END_IF;

		WAIT:
			MpAxisParallel.MoveAbsolute := FALSE;

			IF EDGEPOS(gParallelAxisSettings.diLeft) AND NOT(Saw_SimInputs.diDriveParallelAtFront) THEN
				MpParallelPar.Position := MpAxisParallel.Position + gParallelAxisSettings.aiParallelStep;
				Saw_SimOutputs.aoDriveParallelPosition := Saw_SimOutputs.aoDriveParallelPosition + gParallelAxisSettings.aiParallelStep;

				SMachine := RUNL;
			END_IF;

			IF EDGEPOS(gParallelAxisSettings.diRight) AND NOT(Saw_SimInputs.diDriveParallelAtBack) THEN
				MpParallelPar.Position := MpAxisParallel.Position - gParallelAxisSettings.aiParallelStep;
				Saw_SimOutputs.aoDriveParallelPosition := Saw_SimOutputs.aoDriveParallelPosition - gParallelAxisSettings.aiParallelStep;

				SMachine := RUNR;
			END_IF;

			IF NOT(gParallelAxisSettings.diRunAxis) THEN
				SMachine := INIT;
			END_IF;

		RUNL:
			MpAxisParallel.MoveAbsolute := TRUE;

			IF MpAxisParallel.MoveDone THEN
				SMachine := WAIT;
			END_IF;

		RUNR:
			MpAxisParallel.MoveAbsolute := TRUE;

			IF MpAxisParallel.MoveDone THEN
				SMachine := WAIT;
			END_IF;

	END_CASE;

END_PROGRAM

PROGRAM _EXIT
	(* Insert code here *)

END_PROGRAM
```

### Program Logical/Tasmociag

#### Types.typ
```iecst
TYPE
	StateMachineTyp :
		(
		INIT := 0,
		POWER := 1,
		HOME := 2,
		RUN := 3
		);
END_TYPE
```

#### Variables.var
```iecst
VAR
	SMachine : StateMachineTyp;
	MpConveyorPar : MpAxisBasicParType;
	MpAxisConveyor : MpAxisBasic;
END_VAR
```

#### Main.st
```iecst
PROGRAM _INIT
	MpAxisConveyor.Enable := TRUE;
	MpAxisConveyor.MpLink := ADR(gConveyorAxis);
	MpAxisConveyor.Parameters := ADR(MpConveyorPar);

	SMachine := INIT;

END_PROGRAM

PROGRAM _CYCLIC
	MpAxisConveyor();
	MpConveyorPar.Velocity := gConveyorSettings.aiSpeed;

	CASE SMachine OF
		INIT:
			MpAxisConveyor.Power := FALSE;
			MpAxisConveyor.Home := FALSE;
			MpAxisConveyor.MoveVelocity := FALSE;

			IF EDGEPOS(gConveyorSettings.diActive) AND MpAxisConveyor.Info.ReadyToPowerOn THEN
	  			SMachine := POWER;
			END_IF;

		POWER:
			MpAxisConveyor.Power := TRUE;

			IF MpAxisConveyor.PowerOn THEN
	  			SMachine := HOME;
			END_IF;
		HOME:
			IF NOT(MpAxisConveyor.IsHomed) THEN
				MpAxisConveyor.Home := TRUE;
			END_IF;

			IF MpAxisConveyor.IsHomed THEN
	  			SMachine := RUN;
			END_IF;

		RUN:
			MpAxisConveyor.MoveVelocity := TRUE;

			IF MpAxisConveyor.InVelocity THEN
	  			Saw_SimOutputs.aoTreeVelocity := MpAxisConveyor.Velocity;
			END_IF;

			IF NOT(gConveyorSettings.diActive) THEN
				Saw_SimOutputs.aoTreeVelocity := 0;
				SMachine := INIT;
			END_IF;

	END_CASE;

END_PROGRAM

PROGRAM _EXIT
	(* Insert code here *)

END_PROGRAM
```

Listed in the project but not available here: Logical/Libraries/Saw/Saw_L/MNG_InternalTyp.hpp, Logical/Libraries/Saw/Saw_P/Variables.var, Logical/Libraries/Saw/Types.typ, Logical/MNG_Global.typ
